C07264=1013.290,308.137,352.891,169.642,52.741,160.224
C07265=1013.283,307.846,352.929,169.634,52.748,160.224
C07266=1013.275,307.555,352.966,169.627,52.756,160.225
C07267=1013.269,307.308,352.997,169.621,52.762,160.225
C07268=1013.263,307.060,353.029,169.613,52.768,160.225
C07269=1013.257,306.812,353.061,169.607,52.774,160.225
C07270=1013.251,306.564,353.092,169.600,52.781,160.225
C07271=1013.245,306.316,353.124,169.594,52.787,160.225
C07272=1013.239,306.069,353.155,169.588,52.793,160.225
C07273=1013.233,305.820,353.186,169.581,52.799,160.225
C07274=1013.227,305.573,353.218,169.575,52.805,160.225
C07275=1013.221,305.325,353.250,169.568,52.812,160.226
C07276=1013.214,305.077,353.281,169.562,52.818,160.226
C07277=1013.209,304.829,353.312,169.556,52.824,160.226
C07278=1013.202,304.581,353.343,169.549,52.830,160.226
C07279=1013.197,304.333,353.375,169.543,52.837,160.226
C07280=1013.190,304.085,353.406,169.536,52.843,160.226
C07281=1013.185,303.837,353.437,169.530,52.849,160.227
C07282=1013.178,303.589,353.469,169.524,52.856,160.227
C07283=1013.173,303.342,353.501,169.517,52.862,160.227
C07284=1013.167,303.093,353.531,169.511,52.868,160.227
C07285=1013.161,302.846,353.563,169.505,52.875,160.227
C07286=1013.155,302.597,353.594,169.498,52.881,160.227
C07287=1013.149,302.350,353.625,169.493,52.887,160.228
C07288=1013.144,302.102,353.656,169.486,52.894,160.228
C07289=1013.138,301.854,353.688,169.480,52.900,160.228
C07290=1013.131,301.607,353.719,169.474,52.906,160.228
C07291=1013.126,301.358,353.750,169.467,52.913,160.228
C07292=1013.120,301.110,353.782,169.461,52.919,160.229
C07293=1013.115,300.862,353.812,169.454,52.926,160.229
C07294=1013.109,300.614,353.843,169.448,52.932,160.229
C07295=1013.103,300.366,353.874,169.442,52.938,160.229
C07296=1013.098,300.118,353.905,169.436,52.945,160.230
C07297=1013.091,299.870,353.937,169.430,52.952,160.230
C07298=1013.086,299.622,353.968,169.423,52.958,160.230
C07299=1013.080,299.374,353.998,169.417,52.964,160.230
C07300=1013.074,299.126,354.030,169.411,52.971,160.230
C07301=1013.068,298.878,354.060,169.404,52.977,160.231
C07302=1013.063,298.631,354.092,169.398,52.984,160.231
C07303=1013.057,298.383,354.122,169.393,52.990,160.231
C07304=1013.051,298.134,354.154,169.386,52.997,160.231
C07305=1013.046,297.886,354.184,169.380,53.004,160.232
C07306=1013.040,297.639,354.216,169.373,53.010,160.232
C07307=1013.034,297.391,354.246,169.368,53.017,160.232
C07308=1013.029,297.142,354.277,169.362,53.023,160.232
C07309=1013.023,296.894,354.308,169.355,53.030,160.233
C07310=1013.017,296.647,354.339,169.349,53.037,160.233
C07311=1013.012,296.399,354.370,169.344,53.043,160.233
C07312=1013.007,296.151,354.401,169.337,53.050,160.233
C07313=1013.000,295.902,354.431,169.331,53.056,160.234
C07314=1012.995,295.654,354.462,169.325,53.063,160.234
C07315=1012.989,295.406,354.493,169.318,53.070,160.234
C07316=1012.984,295.158,354.524,169.313,53.076,160.234
C07317=1012.978,294.911,354.554,169.306,53.083,160.235
C07318=1012.973,294.663,354.586,169.300,53.089,160.235
C07319=1012.967,294.415,354.616,169.294,53.096,160.235
C07320=1012.962,294.167,354.647,169.288,53.103,160.235
C07321=1012.956,293.919,354.677,169.282,53.109,160.236
C07322=1012.951,293.671,354.708,169.276,53.116,160.236
C07323=1012.945,293.398,354.742,169.269,53.123,160.236
C07324=1012.939,293.126,354.776,169.262,53.131,160.237
C07325=1012.933,292.853,354.810,169.256,53.138,160.237
C07326=1012.927,292.582,354.843,169.249,53.145,160.237
C07327=1012.922,292.334,354.874,169.243,53.153,160.238
C07328=1012.916,292.085,354.903,169.237,53.159,160.238
C07329=1012.911,291.837,354.934,169.231,53.166,160.238
C07330=1012.905,291.590,354.964,169.225,53.173,160.239
C07331=1012.899,291.342,354.994,169.219,53.180,160.239
C07332=1012.894,291.093,355.024,169.213,53.187,160.239
C07333=1012.888,290.845,355.055,169.207,53.194,160.240
C07334=1012.883,290.597,355.085,169.200,53.201,160.240
C07335=1012.877,290.349,355.115,169.195,53.208,160.240
C07336=1012.871,290.101,355.145,169.189,53.214,160.241
C07337=1012.866,289.853,355.175,169.183,53.222,160.241
C07338=1012.860,289.605,355.205,169.177,53.228,160.241
C07339=1012.854,289.356,355.235,169.171,53.236,160.242
C07340=1012.849,289.109,355.265,169.165,53.242,160.242
C07341=1012.843,288.860,355.295,169.159,53.250,160.242
C07342=1012.837,288.612,355.325,169.153,53.256,160.243
C07343=1012.832,288.364,355.355,169.147,53.264,160.243
C07344=1012.826,288.115,355.384,169.141,53.270,160.243
C07345=1012.821,287.868,355.414,169.135,53.278,160.244
C07346=1012.816,287.620,355.444,169.130,53.285,160.244
C07347=1012.810,287.372,355.474,169.124,53.292,160.245
C07348=1012.804,287.124,355.504,169.118,53.299,160.245
C07349=1012.799,286.875,355.534,169.112,53.306,160.245
C07350=1012.793,286.627,355.564,169.105,53.313,160.246
C07351=1012.787,286.379,355.594,169.100,53.320,160.246
C07352=1012.782,286.131,355.623,169.094,53.328,160.247
C07353=1012.777,285.883,355.653,169.088,53.334,160.247
C07354=1012.771,285.635,355.683,169.082,53.342,160.247
C07355=1012.766,285.386,355.713,169.077,53.349,160.248
C07356=1012.760,285.138,355.742,169.070,53.356,160.248
C07357=1012.755,284.890,355.771,169.065,53.363,160.248
C07358=1012.750,284.642,355.801,169.058,53.371,160.249
C07359=1012.744,284.393,355.831,169.053,53.378,160.249
C07360=1012.738,284.146,355.861,169.047,53.385,160.250
C07361=1012.733,283.898,355.890,169.041,53.392,160.250
C07362=1012.727,283.650,355.919,169.035,53.400,160.250
C07363=1012.722,283.401,355.949,169.029,53.407,160.251
C07364=1012.717,283.154,355.978,169.023,53.414,160.251
C07365=1012.711,282.905,356.007,169.018,53.421,160.252
C07366=1012.705,282.657,356.037,169.012,53.429,160.252
C07367=1012.700,282.408,356.066,169.006,53.436,160.253
C07368=1012.694,282.160,356.095,169.000,53.444,160.253
C07369=1012.689,281.912,356.124,168.995,53.451,160.254
C07370=1012.683,281.664,356.154,168.988,53.459,160.254
C07371=1012.678,281.416,356.183,168.983,53.466,160.255
C07372=1012.672,281.168,356.212,168.977,53.473,160.255
C07373=1012.666,280.919,356.242,168.972,53.481,160.255
C07374=1012.662,280.671,356.270,168.965,53.488,160.256
C07375=1012.656,280.423,356.299,168.960,53.495,160.256
C07376=1012.651,280.175,356.329,168.954,53.503,160.257
C07377=1012.645,279.927,356.358,168.948,53.510,160.257
C07378=1012.640,279.678,356.387,168.942,53.518,160.258
C07379=1012.634,279.430,356.416,168.936,53.525,160.258
C07380=1012.629,279.182,356.445,168.931,53.533,160.259
C07381=1012.624,278.934,356.475,168.924,53.540,160.259
C07382=1012.618,278.685,356.503,168.920,53.548,160.260
C07383=1012.612,278.425,356.534,168.913,53.556,160.260
C07384=1012.607,278.165,356.565,168.907,53.563,160.260
C07385=1012.602,277.905,356.595,168.901,53.572,160.261
C07386=1012.596,277.645,356.626,168.895,53.579,160.261
C07387=1012.587,277.237,356.672,168.886,53.592,160.262
C07388=1012.579,276.829,356.720,168.877,53.604,160.263
C07389=1012.570,276.422,356.768,168.867,53.617,160.264
C07390=1012.561,276.014,356.816,168.858,53.629,160.265
C07391=1012.347,278.241,356.191,168.878,53.661,160.276
C07392=1012.354,278.605,356.149,168.887,53.650,160.276
C07393=1012.362,278.970,356.107,168.895,53.639,160.275
C07394=1012.370,279.335,356.064,168.904,53.628,160.274
C07395=1012.379,279.699,356.021,168.912,53.617,160.274
C07396=1012.383,279.947,355.992,168.918,53.609,160.273
C07397=1012.389,280.196,355.963,168.923,53.602,160.273
C07398=1012.394,280.443,355.934,168.929,53.594,160.272
C07399=1012.400,280.692,355.904,168.936,53.587,160.272
C07400=1012.404,280.940,355.876,168.941,53.580,160.271
C07401=1012.410,281.189,355.846,168.947,53.572,160.271
C07402=1012.416,281.437,355.817,168.952,53.565,160.270
C07403=1012.421,281.684,355.788,168.959,53.557,160.270
C07404=1012.426,281.934,355.759,168.964,53.550,160.270
C07405=1012.433,282.182,355.730,168.970,53.542,160.269
C07406=1012.437,282.429,355.701,168.977,53.535,160.269
C07407=1012.443,282.678,355.671,168.982,53.528,160.268
C07408=1012.448,282.926,355.641,168.988,53.520,160.268
C07409=1012.454,283.174,355.613,168.993,53.513,160.267
C07410=1012.460,283.422,355.583,169.000,53.505,160.267
C07411=1012.465,283.671,355.553,169.005,53.498,160.266
C07412=1012.471,283.918,355.525,169.011,53.490,160.266
C07413=1012.476,284.166,355.495,169.016,53.483,160.266
C07414=1012.482,284.415,355.466,169.023,53.476,160.265
C07415=1012.487,284.663,355.436,169.028,53.469,160.265
C07416=1012.492,284.911,355.407,169.035,53.462,160.264
C07417=1012.498,285.160,355.377,169.040,53.454,160.264
C07418=1012.503,285.408,355.347,169.047,53.447,160.264
C07419=1012.508,285.656,355.318,169.052,53.440,160.263
C07420=1012.514,285.904,355.288,169.058,53.433,160.263
C07421=1012.519,286.152,355.258,169.065,53.425,160.263
C07422=1012.525,286.400,355.228,169.070,53.419,160.262
C07423=1012.530,286.648,355.199,169.077,53.411,160.262
C07424=1012.535,286.897,355.170,169.082,53.404,160.261
C07425=1012.541,287.144,355.139,169.089,53.397,160.261
C07426=1012.547,287.393,355.110,169.094,53.390,160.261
C07427=1012.552,287.641,355.080,169.100,53.382,160.260
C07428=1012.558,287.889,355.050,169.106,53.376,160.260
C07429=1012.563,288.137,355.020,169.112,53.368,160.260
C07430=1012.568,288.385,354.991,169.118,53.362,160.259
C07431=1012.574,288.633,354.960,169.124,53.354,160.259
C07432=1012.580,288.882,354.931,169.129,53.347,160.258
C07433=1012.585,289.130,354.901,169.136,53.340,160.258
C07434=1012.591,289.378,354.871,169.141,53.333,160.258
C07435=1012.597,289.626,354.841,169.148,53.326,160.258
C07436=1012.602,289.874,354.811,169.154,53.319,160.257
C07437=1012.607,290.122,354.781,169.160,53.312,160.257
C07438=1012.613,290.370,354.751,169.166,53.305,160.256
C07439=1012.619,290.618,354.721,169.172,53.298,160.256
C07440=1012.625,290.866,354.691,169.178,53.291,160.256
C07441=1012.630,291.114,354.661,169.183,53.284,160.255
C07442=1012.635,291.362,354.631,169.190,53.277,160.255
C07443=1012.641,291.610,354.600,169.195,53.270,160.255
C07444=1012.646,291.859,354.571,169.202,53.263,160.254
C07445=1012.652,292.107,354.540,169.207,53.256,160.254
C07446=1012.658,292.354,354.510,169.214,53.249,160.254
C07447=1012.663,292.603,354.479,169.220,53.243,160.253
C07448=1012.669,292.877,354.445,169.227,53.235,160.253
C07449=1012.676,293.152,354.412,169.234,53.227,160.253
C07450=1012.681,293.426,354.378,169.240,53.220,160.253
C07451=1012.688,293.701,354.344,169.248,53.213,160.252
C07452=1012.693,293.949,354.313,169.253,53.206,160.252
C07453=1012.699,294.197,354.283,169.259,53.199,160.251
C07454=1012.704,294.445,354.252,169.265,53.192,160.251
C07455=1012.710,294.693,354.221,169.271,53.186,160.251
C07456=1012.715,294.941,354.190,169.278,53.179,160.251
C07457=1012.720,295.189,354.160,169.284,53.172,160.251
C07458=1012.726,295.437,354.129,169.290,53.166,160.250
C07459=1012.731,295.685,354.099,169.296,53.159,160.250
C07460=1012.736,295.933,354.068,169.302,53.153,160.250
C07461=1012.742,296.181,354.037,169.309,53.146,160.250
C07462=1012.747,296.429,354.006,169.314,53.139,160.249
C07463=1012.754,296.677,353.976,169.321,53.132,160.249
C07464=1012.759,296.925,353.944,169.327,53.125,160.249
C07465=1012.765,297.173,353.914,169.332,53.119,160.248
C07466=1012.770,297.421,353.883,169.339,53.112,160.248
C07467=1012.775,297.669,353.852,169.345,53.105,160.248
C07468=1012.781,297.917,353.821,169.352,53.099,160.248
C07469=1012.787,298.165,353.789,169.357,53.092,160.247
C07470=1012.793,298.413,353.759,169.364,53.086,160.247
C07471=1012.798,298.661,353.728,169.370,53.080,160.247
C07472=1012.804,298.909,353.698,169.376,53.073,160.247
C07473=1012.810,299.157,353.666,169.383,53.066,160.247
C07474=1012.815,299.405,353.635,169.389,53.060,160.246
C07475=1012.820,299.653,353.604,169.396,53.053,160.246
C07476=1012.827,299.900,353.573,169.401,53.047,160.246
C07477=1012.832,300.149,353.542,169.407,53.040,160.246
C07478=1012.838,300.397,353.512,169.414,53.033,160.245
C07479=1012.843,300.644,353.480,169.420,53.027,160.245
C07480=1012.850,300.893,353.449,169.427,53.021,160.245
C07481=1012.855,301.140,353.418,169.433,53.014,160.245
C07482=1012.861,301.388,353.387,169.439,53.007,160.245
C07483=1012.867,301.637,353.356,169.445,53.001,160.244
C07484=1012.873,301.884,353.325,169.451,52.995,160.244
C07485=1012.878,302.132,353.294,169.458,52.988,160.244
C07486=1012.885,302.380,353.263,169.464,52.982,160.244
C07487=1012.890,302.628,353.232,169.471,52.976,160.244
C07488=1012.897,302.876,353.200,169.477,52.969,160.244
C07489=1012.902,303.124,353.169,169.484,52.962,160.243
C07490=1012.908,303.372,353.138,169.490,52.956,160.243
C07491=1012.914,303.620,353.106,169.497,52.950,160.243
C07492=1012.920,303.868,353.076,169.503,52.943,160.243
C07493=1012.926,304.116,353.044,169.509,52.938,160.243
C07494=1012.932,304.363,353.013,169.516,52.931,160.243
C07495=1012.937,304.612,352.981,169.521,52.924,160.242
C07496=1012.943,304.859,352.950,169.529,52.918,160.242
C07497=1012.949,305.107,352.918,169.534,52.912,160.242
C07498=1012.955,305.355,352.887,169.542,52.906,160.242
C07499=1012.961,305.603,352.856,169.547,52.899,160.242
C07500=1012.967,305.851,352.824,169.554,52.893,160.242
C07501=1012.973,306.099,352.793,169.560,52.887,160.242
C07502=1012.979,306.348,352.762,169.566,52.880,160.241
C07503=1012.985,306.595,352.730,169.573,52.874,160.241
C07504=1012.991,306.843,352.698,169.579,52.868,160.241
C07505=1012.997,307.090,352.667,169.586,52.862,160.241
C07506=1013.003,307.338,352.635,169.593,52.856,160.241
C07507=1013.010,307.587,352.605,169.599,52.849,160.241
C07508=1013.016,307.879,352.566,169.607,52.842,160.241
C07509=1013.024,308.172,352.530,169.615,52.835,160.241
C07510=1013.031,308.464,352.493,169.623,52.828,160.240
C07511=1013.038,308.757,352.456,169.630,52.820,160.240
C07512=1013.044,309.004,352.423,169.636,52.814,160.240
C07513=1013.050,309.252,352.391,169.643,52.808,160.240
C07514=1013.056,309.501,352.359,169.650,52.802,160.240
C07515=1013.061,309.748,352.327,169.656,52.796,160.240
C07516=1013.068,309.996,352.295,169.663,52.790,160.240
C07517=1013.072,310.244,352.262,169.669,52.784,160.240
C07518=1013.079,310.491,352.230,169.675,52.778,160.240
C07519=1013.085,310.739,352.198,169.683,52.772,160.240
C07520=1013.090,310.987,352.166,169.689,52.766,160.240
C07521=1013.096,311.235,352.133,169.695,52.761,160.239
C07522=1013.102,311.483,352.101,169.702,52.754,160.239
C07523=1013.108,311.731,352.068,169.709,52.749,160.239
C07524=1013.113,311.978,352.036,169.715,52.743,160.239
C07525=1013.120,312.226,352.004,169.722,52.737,160.239
C07526=1013.126,312.474,351.971,169.728,52.731,160.239
C07527=1013.132,312.722,351.939,169.735,52.725,160.239
C07528=1013.137,312.969,351.907,169.742,52.719,160.239
C07529=1013.143,313.217,351.874,169.748,52.714,160.239
C07530=1013.149,313.465,351.841,169.755,52.708,160.239
C07531=1013.155,313.713,351.809,169.762,52.702,160.239
C07532=1013.161,313.960,351.776,169.768,52.696,160.239
C07533=1013.168,314.208,351.743,169.775,52.690,160.239
C07534=1013.173,314.455,351.712,169.781,52.684,160.239
C07535=1013.179,314.703,351.678,169.789,52.678,160.239
C07536=1013.185,314.951,351.646,169.795,52.673,160.239
C07537=1013.191,315.199,351.614,169.802,52.667,160.239
C07538=1013.197,315.447,351.581,169.809,52.661,160.239
C07539=1013.203,315.694,351.548,169.815,52.656,160.239
C07540=1013.209,315.942,351.515,169.821,52.650,160.239
C07541=1013.215,316.190,351.483,169.829,52.644,160.239
C07542=1013.221,316.438,351.450,169.835,52.639,160.239
C07543=1013.228,316.686,351.417,169.842,52.633,160.239
C07544=1013.234,316.933,351.385,169.849,52.627,160.239
C07545=1013.240,317.181,351.352,169.855,52.622,160.239
C07546=1013.246,317.429,351.319,169.863,52.616,160.239
C07547=1013.252,317.677,351.287,169.869,52.610,160.239
C07548=1013.258,317.925,351.254,169.877,52.605,160.239
C07549=1013.264,318.172,351.221,169.883,52.599,160.239
C07550=1013.271,318.420,351.188,169.890,52.593,160.239
C07551=1013.276,318.668,351.155,169.897,52.588,160.239
C07552=1013.282,318.915,351.122,169.903,52.582,160.239
C07553=1013.289,319.163,351.089,169.910,52.576,160.239
C07554=1013.296,319.411,351.056,169.917,52.571,160.239
C07555=1013.302,319.659,351.024,169.924,52.565,160.239
C07556=1013.307,319.907,350.990,169.931,52.560,160.240
C07557=1013.314,320.154,350.958,169.937,52.554,160.239
C07558=1013.320,320.401,350.924,169.945,52.549,160.240
C07559=1013.327,320.649,350.891,169.951,52.543,160.240
C07560=1013.334,320.897,350.858,169.959,52.538,160.240
C07561=1013.339,321.145,350.825,169.965,52.532,160.240
C07562=1013.345,321.393,350.792,169.973,52.526,160.240
C07563=1013.352,321.640,350.759,169.979,52.521,160.240
C07564=1013.359,321.888,350.726,169.987,52.515,160.240
C07565=1013.365,322.135,350.693,169.993,52.510,160.240
C07566=1013.371,322.383,350.660,170.000,52.505,160.240
C07567=1013.377,322.631,350.627,170.007,52.499,160.240
C07568=1013.385,322.929,350.587,170.016,52.493,160.241
C07569=1013.393,323.227,350.547,170.024,52.486,160.241
C07570=1013.401,323.525,350.507,170.032,52.480,160.241
C07571=1013.409,323.824,350.467,170.041,52.473,160.241
C07572=1013.415,324.072,350.433,170.048,52.468,160.241
C07573=1013.421,324.319,350.400,170.055,52.462,160.241
C07574=1013.428,324.567,350.367,170.062,52.457,160.241
C07575=1013.435,324.814,350.334,170.070,52.451,160.241
C07576=1013.441,325.061,350.301,170.076,52.446,160.242
C07577=1013.447,325.310,350.267,170.083,52.441,160.241
C07578=1013.454,325.557,350.233,170.090,52.435,160.242
C07579=1013.461,325.805,350.200,170.097,52.430,160.242
C07580=1013.467,326.053,350.166,170.105,52.425,160.242
C07581=1013.473,326.300,350.132,170.112,52.420,160.242
C07582=1013.480,326.548,350.098,170.119,52.414,160.242
C07583=1013.486,326.795,350.064,170.126,52.409,160.243
C07584=1013.493,327.043,350.031,170.133,52.404,160.243
C07585=1013.498,327.290,349.997,170.140,52.399,160.243
C07586=1013.505,327.538,349.963,170.147,52.394,160.243
C07587=1013.511,327.785,349.929,170.155,52.389,160.243
C07588=1013.518,328.033,349.895,170.161,52.384,160.243
C07589=1013.524,328.281,349.861,170.169,52.378,160.244
C07590=1013.531,328.528,349.827,170.176,52.373,160.244
C07591=1013.537,328.776,349.793,170.183,52.369,160.244
C07592=1013.543,329.024,349.758,170.191,52.363,160.244
C07593=1013.551,329.271,349.725,170.197,52.358,160.244
C07594=1013.556,329.519,349.691,170.205,52.353,160.245
C07595=1013.563,329.767,349.656,170.212,52.348,160.245
C07596=1013.569,330.014,349.623,170.219,52.343,160.245
C07597=1013.576,330.262,349.588,170.227,52.338,160.245
C07598=1013.582,330.509,349.554,170.234,52.333,160.246
C07599=1013.589,330.756,349.520,170.241,52.328,160.246
C07600=1013.595,331.004,349.486,170.249,52.322,160.246
C07601=1013.602,331.252,349.452,170.256,52.318,160.246
C07602=1013.609,331.499,349.417,170.264,52.313,160.247
C07603=1013.615,331.747,349.383,170.270,52.308,160.247
C07604=1013.622,331.995,349.349,170.277,52.303,160.247
C07605=1013.628,332.243,349.314,170.285,52.298,160.247
C07606=1013.635,332.489,349.280,170.292,52.294,160.248
C07607=1013.642,332.737,349.246,170.300,52.288,160.248
C07608=1013.648,332.984,349.210,170.307,52.283,160.248
C07609=1013.655,333.232,349.176,170.315,52.279,160.248
C07610=1013.661,333.480,349.142,170.321,52.274,160.248
C07611=1013.667,333.727,349.107,170.330,52.269,160.249
C07612=1013.674,333.975,349.072,170.337,52.264,160.249
C07613=1013.681,334.222,349.037,170.344,52.259,160.249
C07614=1013.687,334.470,349.003,170.352,52.255,160.250
C07615=1013.694,334.718,348.968,170.358,52.250,160.250
C07616=1013.700,334.964,348.933,170.366,52.245,160.250
C07617=1013.707,335.212,348.899,170.373,52.240,160.250
C07618=1013.714,335.459,348.864,170.381,52.235,160.251
C07619=1013.720,335.707,348.830,170.388,52.231,160.251
C07620=1013.727,335.955,348.794,170.396,52.226,160.251
C07621=1013.734,336.202,348.759,170.403,52.221,160.252
C07622=1013.740,336.450,348.725,170.411,52.217,160.252
C07623=1013.747,336.698,348.690,170.418,52.212,160.253
C07624=1013.754,336.945,348.655,170.426,52.207,160.253
C07625=1013.761,337.192,348.619,170.433,52.202,160.253
C07626=1013.768,337.440,348.584,170.441,52.198,160.254
C07627=1013.774,337.688,348.550,170.449,52.193,160.254
C07628=1013.782,337.981,348.509,170.458,52.187,160.254
C07629=1013.790,338.275,348.467,170.467,52.182,160.255
C07630=1013.798,338.568,348.425,170.476,52.176,160.255
C07631=1013.807,338.863,348.383,170.485,52.171,160.256
C07632=1013.813,339.110,348.348,170.492,52.167,160.256
C07633=1013.819,339.358,348.312,170.500,52.162,160.256
C07634=1013.826,339.605,348.277,170.507,52.157,160.257
C07635=1013.833,339.852,348.242,170.515,52.153,160.257
C07636=1013.840,340.100,348.207,170.522,52.148,160.257
C07637=1013.847,340.347,348.172,170.531,52.144,160.258
C07638=1013.854,340.594,348.136,170.538,52.140,160.258
C07639=1013.860,340.842,348.100,170.546,52.135,160.259
C07640=1013.867,341.090,348.065,170.554,52.130,160.259
C07641=1013.874,341.337,348.030,170.562,52.126,160.260
C07642=1013.881,341.584,347.994,170.570,52.121,160.260
C07643=1013.888,341.831,347.959,170.577,52.117,160.260
C07644=1013.894,342.079,347.923,170.585,52.112,160.261
C07645=1013.901,342.326,347.887,170.593,52.109,160.261
C07646=1013.908,342.574,347.852,170.601,52.104,160.262
C07647=1013.915,342.821,347.816,170.608,52.100,160.262
C07648=1013.922,343.069,347.780,170.616,52.095,160.262
C07649=1013.929,343.316,347.744,170.624,52.091,160.263
C07650=1013.936,343.563,347.709,170.632,52.086,160.263
C07651=1013.942,343.810,347.673,170.640,52.082,160.264
C07652=1013.949,344.058,347.637,170.647,52.078,160.264
C07653=1013.956,344.305,347.602,170.656,52.073,160.265
C07654=1013.963,344.552,347.566,170.663,52.069,160.265
C07655=1013.971,344.799,347.529,170.671,52.065,160.266
C07656=1013.977,345.047,347.494,170.678,52.061,160.266
C07657=1013.985,345.295,347.458,170.686,52.056,160.267
C07658=1013.992,345.541,347.422,170.695,52.052,160.267
C07659=1013.998,345.789,347.387,170.702,52.048,160.268
C07660=1014.005,346.036,347.350,170.711,52.044,160.268
C07661=1014.012,346.283,347.314,170.718,52.039,160.269
C07662=1014.020,346.531,347.278,170.726,52.035,160.269
C07663=1014.026,346.778,347.242,170.735,52.030,160.270
C07664=1014.034,347.026,347.206,170.742,52.027,160.270
C07665=1014.040,347.273,347.169,170.751,52.023,160.271
C07666=1014.048,347.520,347.133,170.758,52.018,160.271
C07667=1014.054,347.767,347.097,170.766,52.014,160.272
C07668=1014.062,348.015,347.060,170.775,52.010,160.272
C07669=1014.068,348.262,347.024,170.782,52.006,160.273
C07670=1014.076,348.509,346.988,170.791,52.002,160.273
C07671=1014.082,348.756,346.951,170.799,51.998,160.274
C07672=1014.090,349.004,346.915,170.807,51.994,160.275
C07673=1014.097,349.251,346.878,170.815,51.989,160.275
C07674=1014.104,349.498,346.842,170.823,51.986,160.276
C07675=1014.111,349.745,346.805,170.831,51.982,160.276
C07676=1014.118,349.992,346.769,170.840,51.978,160.277
C07677=1014.125,350.240,346.732,170.847,51.974,160.277
C07678=1014.133,350.487,346.695,170.856,51.970,160.278
C07679=1014.139,350.734,346.659,170.864,51.966,160.279
C07680=1014.147,350.981,346.623,170.871,51.962,160.279
C07681=1014.154,351.229,346.586,170.880,51.958,160.280
C07682=1014.161,351.476,346.548,170.889,51.954,160.280
C07683=1014.168,351.723,346.512,170.896,51.950,160.281
C07684=1014.175,351.971,346.476,170.905,51.946,160.281
C07685=1014.183,352.217,346.439,170.913,51.942,160.282
C07686=1014.190,352.465,346.402,170.922,51.938,160.283
C07687=1014.198,352.711,346.365,170.929,51.934,160.283
C07688=1014.206,353.003,346.321,170.940,51.929,160.284
C07689=1014.215,353.294,346.278,170.950,51.925,160.285
C07690=1014.223,353.586,346.234,170.959,51.920,160.286
C07691=1014.232,353.877,346.191,170.969,51.916,160.286
C07692=1014.239,354.124,346.154,170.978,51.913,160.287
C07693=1014.246,354.372,346.117,170.986,51.908,160.288
C07694=1014.254,354.618,346.080,170.994,51.905,160.288
C07695=1014.261,354.865,346.043,171.002,51.901,160.289
C07696=1014.268,355.112,346.005,171.011,51.897,160.290
C07697=1014.275,355.359,345.968,171.020,51.893,160.290
C07698=1014.283,355.607,345.931,171.027,51.890,160.291
C07699=1014.290,355.854,345.894,171.036,51.886,160.292
C07700=1014.298,356.101,345.856,171.045,51.882,160.292
C07701=1014.306,356.348,345.819,171.053,51.878,160.293
C07702=1014.313,356.595,345.782,171.061,51.875,160.294
C07703=1014.320,356.842,345.744,171.070,51.871,160.294
C07704=1014.327,357.089,345.707,171.079,51.868,160.295
C07705=1014.335,357.336,345.669,171.088,51.864,160.296
C07706=1014.343,357.583,345.632,171.097,51.860,160.297
C07707=1014.350,357.831,345.595,171.104,51.857,160.297
C07708=1014.358,358.078,345.557,171.113,51.853,160.298
C07709=1014.365,358.325,345.519,171.122,51.850,160.299
C07710=1014.373,358.571,345.482,171.131,51.846,160.300
C07711=1014.380,358.818,345.444,171.140,51.842,160.301
C07712=1014.388,359.066,345.407,171.147,51.839,160.301
C07713=1014.395,359.312,345.369,171.156,51.835,160.302
C07714=1014.402,359.559,345.331,171.165,51.832,160.303
C07715=1014.410,359.807,345.293,171.174,51.828,160.304
C07716=1014.417,360.054,345.254,171.183,51.824,160.304
C07717=1014.424,360.301,345.217,171.191,51.821,160.305
C07718=1014.432,360.548,345.179,171.200,51.818,160.306
C07719=1014.439,360.795,345.141,171.209,51.815,160.307
C07720=1014.447,361.042,345.102,171.218,51.811,160.308
C07721=1014.455,361.289,345.065,171.227,51.808,160.308
C07722=1014.462,361.536,345.027,171.236,51.804,160.309
C07723=1014.470,361.782,344.988,171.243,51.801,160.310
C07724=1014.478,362.030,344.950,171.252,51.797,160.311
C07725=1014.485,362.276,344.912,171.261,51.794,160.311
C07726=1014.493,362.523,344.874,171.270,51.790,160.312
C07727=1014.500,362.771,344.836,171.279,51.787,160.313
C07728=1014.508,363.017,344.798,171.288,51.784,160.314
C07729=1014.516,363.264,344.759,171.297,51.780,160.315
C07730=1014.524,363.511,344.721,171.306,51.777,160.316
C07731=1014.531,363.758,344.683,171.315,51.774,160.317
C07732=1014.539,364.005,344.645,171.324,51.771,160.318
C07733=1014.547,364.252,344.607,171.332,51.768,160.318
C07734=1014.555,364.499,344.568,171.341,51.764,160.319
C07735=1014.562,364.746,344.530,171.350,51.761,160.320
C07736=1014.571,364.993,344.491,171.359,51.757,160.321
C07737=1014.578,365.239,344.453,171.369,51.755,160.322
C07738=1014.586,365.487,344.414,171.378,51.751,160.323
C07739=1014.593,365.733,344.375,171.387,51.748,160.324
C07740=1014.601,365.981,344.337,171.396,51.745,160.325
C07741=1014.609,366.228,344.298,171.405,51.742,160.325
C07742=1014.617,366.474,344.260,171.414,51.738,160.326
C07743=1014.625,366.722,344.221,171.423,51.735,160.327
C07744=1014.633,366.967,344.182,171.432,51.732,160.328
C07745=1014.641,367.215,344.144,171.441,51.729,160.329
C07746=1014.649,367.462,344.105,171.451,51.726,160.330
C07747=1014.656,367.708,344.066,171.460,51.722,160.331
C07748=1014.666,368.007,344.019,171.471,51.719,160.332
C07749=1014.675,368.306,343.971,171.482,51.715,160.333
C07750=1014.685,368.605,343.925,171.494,51.712,160.335
C07751=1014.694,368.903,343.876,171.505,51.708,160.336
C07752=1014.702,369.151,343.838,171.514,51.705,160.337
C07753=1014.711,369.397,343.798,171.524,51.702,160.338
C07754=1014.718,369.643,343.759,171.533,51.699,160.339
C07755=1014.726,369.891,343.720,171.542,51.696,160.340
C07756=1014.734,370.138,343.680,171.551,51.693,160.341
C07757=1014.742,370.384,343.641,171.561,51.690,160.342
C07758=1014.750,370.631,343.602,171.570,51.688,160.343
C07759=1014.758,370.878,343.562,171.580,51.684,160.344
C07760=1014.766,371.124,343.524,171.590,51.681,160.345
C07761=1014.775,371.371,343.484,171.599,51.678,160.346
C07762=1014.782,371.618,343.444,171.608,51.676,160.347
C07763=1014.790,371.865,343.406,171.618,51.673,160.348
C07764=1014.798,372.112,343.366,171.627,51.670,160.349
C07765=1014.807,372.358,343.326,171.636,51.667,160.350
C07766=1014.815,372.605,343.287,171.646,51.664,160.351
C07767=1014.823,372.852,343.247,171.656,51.661,160.352
C07768=1014.831,373.099,343.208,171.666,51.658,160.353
C07769=1014.840,373.345,343.169,171.675,51.656,160.354
C07770=1014.847,373.592,343.129,171.684,51.653,160.356
C07771=1014.856,373.838,343.089,171.694,51.650,160.357
C07772=1014.864,374.085,343.049,171.704,51.647,160.358
C07773=1014.872,374.331,343.009,171.714,51.644,160.359
C07774=1014.881,374.578,342.970,171.723,51.642,160.360
C07775=1014.889,374.826,342.930,171.733,51.639,160.361
C07776=1014.898,375.072,342.890,171.743,51.636,160.362
C07777=1014.906,375.319,342.850,171.753,51.633,160.363
C07778=1014.914,375.565,342.810,171.762,51.631,160.365
C07779=1014.922,375.811,342.770,171.772,51.628,160.366
C07780=1014.930,376.058,342.730,171.782,51.625,160.367
C07781=1014.939,376.305,342.689,171.792,51.623,160.368
C07782=1014.947,376.552,342.650,171.801,51.620,160.369
C07783=1014.955,376.798,342.609,171.811,51.618,160.370
C07784=1014.963,377.044,342.568,171.822,51.615,160.372
C07785=1014.971,377.291,342.529,171.831,51.613,160.373
C07786=1014.980,377.538,342.488,171.841,51.610,160.374
C07787=1014.988,377.784,342.447,171.852,51.607,160.375
C07788=1014.997,378.030,342.407,171.861,51.605,160.376
C07789=1015.005,378.278,342.367,171.871,51.603,160.378
C07790=1015.013,378.524,342.326,171.882,51.600,160.379
C07791=1015.021,378.771,342.286,171.891,51.598,160.380
C07792=1015.031,379.017,342.245,171.901,51.595,160.381
C07793=1015.039,379.263,342.205,171.911,51.592,160.383
C07794=1015.047,379.510,342.164,171.921,51.590,160.384
C07795=1015.056,379.756,342.124,171.931,51.588,160.385
C07796=1015.064,380.003,342.083,171.941,51.585,160.386
C07797=1015.073,380.250,342.042,171.951,51.583,160.387
C07798=1015.081,380.496,342.001,171.962,51.580,160.389
C07799=1015.090,380.743,341.961,171.972,51.578,160.390
C07800=1015.098,380.989,341.920,171.983,51.576,160.391
C07801=1015.107,381.236,341.879,171.992,51.573,160.393
C07802=1015.116,381.482,341.838,172.002,51.571,160.394
C07803=1015.124,381.728,341.798,172.013,51.569,160.395
C07804=1015.133,381.975,341.757,172.023,51.567,160.397
C07805=1015.141,382.222,341.716,172.034,51.564,160.398
C07806=1015.151,382.468,341.675,172.043,51.562,160.399
C07807=1015.159,382.715,341.634,172.054,51.559,160.401
C07808=1015.170,383.036,341.580,172.067,51.557,160.402
C07809=1015.182,383.357,341.527,172.082,51.553,160.404
C07810=1015.193,383.679,341.473,172.095,51.551,160.406
C07811=1015.205,384.000,341.420,172.109,51.547,160.408
C07812=1015.214,384.247,341.379,172.119,51.546,160.409
C07813=1015.223,384.494,341.338,172.130,51.543,160.410
C07814=1015.232,384.740,341.296,172.140,51.540,160.412
C07815=1015.241,384.987,341.254,172.151,51.539,160.413
C07816=1015.249,385.232,341.213,172.161,51.536,160.415
C07817=1015.258,385.479,341.172,172.172,51.535,160.416
C07818=1015.267,385.726,341.130,172.182,51.532,160.417
C07819=1015.276,385.972,341.088,172.194,51.530,160.419
C07820=1015.284,386.218,341.047,172.203,51.528,160.420
C07821=1015.293,386.465,341.005,172.215,51.526,160.422
C07822=1015.303,386.711,340.964,172.225,51.524,160.423
C07823=1015.312,386.957,340.922,172.236,51.522,160.425
C07824=1015.321,387.203,340.880,172.247,51.520,160.426
C07825=1015.330,387.450,340.839,172.258,51.517,160.428
C07826=1015.339,387.696,340.797,172.268,51.516,160.429
C07827=1015.347,387.942,340.754,172.279,51.514,160.431
C07828=1015.356,388.189,340.712,172.290,51.512,160.432
C07829=1015.365,388.435,340.671,172.301,51.509,160.434
C07830=1015.374,388.681,340.629,172.311,51.508,160.435
C07831=1015.383,388.927,340.586,172.322,51.506,160.437
C07832=1015.392,389.173,340.545,172.334,51.504,160.438
C07833=1015.401,389.419,340.502,172.345,51.502,160.440
C07834=1015.410,389.665,340.461,172.355,51.500,160.441
C07835=1015.420,389.911,340.418,172.366,51.498,160.443
C07836=1015.428,390.159,340.375,172.377,51.497,160.444
C07837=1015.438,390.404,340.333,172.389,51.495,160.446
C07838=1015.447,390.651,340.291,172.400,51.493,160.448
C07839=1015.456,390.896,340.249,172.411,51.491,160.449
C07840=1015.466,391.143,340.206,172.423,51.489,160.451
C07841=1015.475,391.389,340.164,172.433,51.488,160.452
C07842=1015.484,391.635,340.122,172.444,51.486,160.454
C07843=1015.494,391.881,340.079,172.455,51.484,160.456
C07844=1015.502,392.128,340.036,172.466,51.482,160.457
C07845=1015.511,392.374,339.994,172.478,51.480,160.459
C07846=1015.521,392.620,339.952,172.489,51.479,160.460
C07847=1015.530,392.866,339.909,172.501,51.477,160.462
C07848=1015.539,393.112,339.866,172.512,51.475,160.464
C07849=1015.549,393.358,339.823,172.523,51.473,160.465
C07850=1015.557,393.604,339.780,172.535,51.472,160.467
C07851=1015.567,393.850,339.737,172.546,51.470,160.469
C07852=1015.576,394.096,339.694,172.558,51.469,160.470
C07853=1015.586,394.343,339.652,172.569,51.467,160.472
C07854=1015.595,394.589,339.609,172.581,51.465,160.474
C07855=1015.605,394.835,339.565,172.592,51.464,160.476
C07856=1015.614,395.080,339.523,172.604,51.462,160.477
C07857=1015.623,395.327,339.479,172.615,51.460,160.479
C07858=1015.633,395.573,339.436,172.627,51.459,160.481
C07859=1015.643,395.819,339.393,172.638,51.458,160.483
C07860=1015.653,396.065,339.350,172.650,51.456,160.484
C07861=1015.662,396.311,339.306,172.661,51.454,160.486
C07862=1015.671,396.557,339.264,172.674,51.453,160.488
C07863=1015.681,396.803,339.220,172.685,51.451,160.490
C07864=1015.691,397.049,339.176,172.697,51.450,160.491
C07865=1015.700,397.295,339.134,172.708,51.449,160.493
C07866=1015.709,397.541,339.090,172.720,51.447,160.495
C07867=1015.720,397.787,339.046,172.732,51.446,160.497
C07868=1015.736,398.202,338.973,172.752,51.443,160.500
C07869=1015.751,398.617,338.899,172.772,51.441,160.503
C07870=1015.398,396.589,338.913,172.658,51.516,160.502
C07871=1015.388,396.343,338.956,172.647,51.518,160.501
C07872=1015.379,396.096,339.000,172.635,51.520,160.499
C07873=1015.369,395.851,339.043,172.622,51.522,160.497
C07874=1015.359,395.605,339.086,172.611,51.523,160.495
C07875=1015.349,395.359,339.129,172.600,51.525,160.494
C07876=1015.341,395.113,339.172,172.588,51.526,160.492
C07877=1015.331,394.867,339.215,172.577,51.528,160.490
C07878=1015.322,394.621,339.257,172.565,51.530,160.488
C07879=1015.312,394.375,339.301,172.554,51.531,160.487
C07880=1015.303,394.129,339.344,172.542,51.533,160.485
C07881=1015.293,393.883,339.387,172.531,51.534,160.483
C07882=1015.284,393.637,339.429,172.519,51.537,160.482
C07883=1015.275,393.390,339.472,172.507,51.539,160.480
C07884=1015.266,393.144,339.515,172.496,51.540,160.478
C07885=1015.256,392.899,339.557,172.484,51.542,160.477
C07886=1015.247,392.652,339.601,172.473,51.544,160.475
C07887=1015.238,392.406,339.643,172.462,51.545,160.473
C07888=1015.229,392.160,339.686,172.450,51.547,160.472
C07889=1015.219,391.914,339.728,172.439,51.549,160.470
C07890=1015.211,391.667,339.771,172.429,51.550,160.468
C07891=1015.201,391.421,339.813,172.417,51.552,160.467
C07892=1015.192,391.175,339.856,172.406,51.554,160.465
C07893=1015.183,390.929,339.898,172.395,51.556,160.464
C07894=1015.173,390.683,339.940,172.384,51.558,160.462
C07895=1015.164,390.437,339.983,172.373,51.560,160.461
C07896=1015.155,390.190,340.025,172.361,51.562,160.459
C07897=1015.145,389.944,340.067,172.350,51.564,160.457
C07898=1015.137,389.698,340.109,172.339,51.566,160.456
C07899=1015.128,389.452,340.152,172.328,51.568,160.454
C07900=1015.119,389.206,340.194,172.317,51.570,160.453
C07901=1015.110,388.959,340.235,172.307,51.572,160.451
C07902=1015.101,388.713,340.278,172.296,51.574,160.450
C07903=1015.092,388.467,340.319,172.284,51.576,160.448
C07904=1015.083,388.221,340.361,172.273,51.578,160.447
C07905=1015.074,387.974,340.403,172.262,51.580,160.445
C07906=1015.065,387.729,340.445,172.252,51.582,160.444
C07907=1015.056,387.482,340.487,172.241,51.584,160.442
C07908=1015.047,387.236,340.529,172.230,51.586,160.441
C07909=1015.038,386.989,340.570,172.219,51.589,160.439
C07910=1015.029,386.743,340.612,172.209,51.590,160.438
C07911=1015.020,386.497,340.654,172.198,51.593,160.436
C07912=1015.011,386.250,340.696,172.187,51.595,160.435
C07913=1015.002,386.004,340.737,172.176,51.598,160.434
C07914=1014.993,385.758,340.779,172.166,51.599,160.432
C07915=1014.985,385.511,340.820,172.155,51.602,160.431
C07916=1014.976,385.265,340.861,172.144,51.604,160.429
C07917=1014.968,385.019,340.903,172.134,51.606,160.428
C07918=1014.959,384.772,340.945,172.123,51.608,160.426
C07919=1014.950,384.525,340.986,172.112,51.611,160.425
C07920=1014.941,384.279,341.027,172.102,51.613,160.424
C07921=1014.932,384.033,341.068,172.091,51.615,160.422
C07922=1014.923,383.787,341.109,172.081,51.618,160.421
C07923=1014.915,383.537,341.151,172.071,51.620,160.420
C07924=1014.906,383.289,341.191,172.060,51.622,160.418
C07925=1014.897,383.040,341.234,172.049,51.625,160.417
C07926=1014.888,382.792,341.274,172.039,51.627,160.415
C07927=1014.879,382.545,341.315,172.028,51.629,160.414
C07928=1014.871,382.299,341.357,172.018,51.631,160.413
C07929=1014.862,382.052,341.398,172.008,51.634,160.411
C07930=1014.853,381.806,341.438,171.997,51.636,160.410
C07931=1014.845,381.559,341.479,171.987,51.639,160.409
C07932=1014.836,381.312,341.520,171.977,51.642,160.408
C07933=1014.827,381.067,341.561,171.967,51.644,160.406
C07934=1014.818,380.820,341.602,171.956,51.646,160.405
C07935=1014.810,380.574,341.642,171.946,51.649,160.404
C07936=1014.801,380.327,341.683,171.935,51.651,160.402
C07937=1014.793,380.081,341.723,171.926,51.653,160.401
C07938=1014.784,379.834,341.764,171.915,51.657,160.400
C07939=1014.776,379.587,341.805,171.905,51.659,160.399
C07940=1014.767,379.341,341.845,171.895,51.661,160.397
C07941=1014.759,379.094,341.886,171.885,51.664,160.396
C07942=1014.751,378.848,341.927,171.875,51.666,160.395
C07943=1014.742,378.601,341.966,171.865,51.669,160.394
C07944=1014.734,378.355,342.007,171.855,51.672,160.393
C07945=1014.726,378.108,342.048,171.844,51.674,160.391
C07946=1014.717,377.861,342.089,171.835,51.677,160.390
C07947=1014.709,377.615,342.128,171.825,51.679,160.389
C07948=1014.701,377.368,342.169,171.815,51.682,160.388
C07949=1014.693,377.122,342.209,171.805,51.684,160.386
C07950=1014.684,376.875,342.249,171.796,51.687,160.385
C07951=1014.676,376.629,342.289,171.785,51.690,160.384
C07952=1014.667,376.382,342.330,171.775,51.693,160.383
C07953=1014.660,376.135,342.370,171.766,51.695,160.382
C07954=1014.651,375.889,342.410,171.755,51.698,160.381
C07955=1014.643,375.643,342.450,171.746,51.701,160.380
C07956=1014.635,375.396,342.491,171.736,51.704,160.378
C07957=1014.626,375.149,342.530,171.726,51.706,160.377
C07958=1014.618,374.902,342.570,171.716,51.709,160.376
C07959=1014.610,374.655,342.610,171.707,51.712,160.375
C07960=1014.602,374.409,342.649,171.697,51.715,160.374
C07961=1014.594,374.163,342.690,171.687,51.718,160.373
C07962=1014.585,373.916,342.729,171.678,51.720,160.372
C07963=1014.577,373.669,342.768,171.668,51.723,160.371
C07964=1014.569,373.422,342.808,171.658,51.726,160.370
C07965=1014.560,373.176,342.847,171.649,51.729,160.368
C07966=1014.553,372.929,342.887,171.639,51.732,160.367
C07967=1014.544,372.682,342.927,171.630,51.735,160.366
C07968=1014.536,372.436,342.966,171.619,51.738,160.365
C07969=1014.528,372.189,343.006,171.610,51.741,160.364
C07970=1014.520,371.942,343.045,171.601,51.744,160.363
C07971=1014.511,371.695,343.084,171.591,51.746,160.362
C07972=1014.504,371.448,343.124,171.581,51.749,160.361
C07973=1014.495,371.202,343.163,171.572,51.753,160.360
C07974=1014.488,370.955,343.203,171.562,51.756,160.359
C07975=1014.479,370.708,343.242,171.553,51.758,160.358
C07976=1014.472,370.462,343.281,171.544,51.761,160.357
C07977=1014.464,370.215,343.320,171.535,51.765,160.356
C07978=1014.455,369.968,343.360,171.525,51.767,160.355
C07979=1014.447,369.721,343.398,171.515,51.771,160.354
C07980=1014.440,369.475,343.438,171.506,51.774,160.353
C07981=1014.432,369.227,343.477,171.497,51.777,160.352
C07982=1014.424,368.980,343.517,171.487,51.780,160.351
C07983=1014.415,368.680,343.564,171.476,51.784,160.350
C07984=1014.405,368.378,343.611,171.465,51.787,160.349
C07985=1014.396,368.077,343.659,171.453,51.791,160.347
C07986=1014.386,367.776,343.707,171.442,51.795,160.346
C07987=1014.378,367.530,343.746,171.433,51.798,160.345
C07988=1014.371,367.283,343.785,171.424,51.801,160.344
C07989=1014.362,367.035,343.823,171.415,51.804,160.343
C07990=1014.355,366.789,343.862,171.405,51.808,160.342
C07991=1014.346,366.542,343.901,171.396,51.811,160.341
C07992=1014.339,366.296,343.939,171.387,51.815,160.341
C07993=1014.331,366.049,343.978,171.377,51.817,160.340
C07994=1014.323,365.801,344.016,171.368,51.821,160.339
C07995=1014.315,365.555,344.055,171.359,51.824,160.338
C07996=1014.307,365.308,344.093,171.350,51.828,160.337
C07997=1014.299,365.061,344.131,171.341,51.831,160.336
C07998=1014.291,364.814,344.170,171.332,51.834,160.335
C07999=1014.284,364.567,344.209,171.323,51.837,160.334
C08000=1014.276,364.320,344.248,171.314,51.841,160.333
C08001=1014.269,364.073,344.285,171.305,51.844,160.333
C08002=1014.261,363.826,344.323,171.296,51.848,160.332
C08003=1014.253,363.579,344.362,171.287,51.851,160.331
C08004=1014.246,363.332,344.400,171.278,51.854,160.330
C08005=1014.238,363.085,344.439,171.269,51.858,160.329
C08006=1014.230,362.838,344.476,171.260,51.861,160.328
C08007=1014.223,362.592,344.515,171.251,51.865,160.327
C08008=1014.215,362.344,344.553,171.242,51.868,160.327
C08009=1014.207,362.097,344.591,171.233,51.872,160.326
C08010=1014.200,361.851,344.629,171.224,51.875,160.325
C08011=1014.192,361.603,344.667,171.215,51.878,160.324
C08012=1014.184,361.356,344.705,171.208,51.882,160.324
C08013=1014.177,361.110,344.743,171.199,51.885,160.323
C08014=1014.170,360.863,344.781,171.190,51.889,160.322
C08015=1014.161,360.615,344.819,171.181,51.892,160.321
C08016=1014.154,360.368,344.857,171.172,51.896,160.320
C08017=1014.147,360.121,344.894,171.163,51.900,160.319
C08018=1014.139,359.875,344.933,171.154,51.903,160.319
C08019=1014.132,359.628,344.970,171.145,51.907,160.318
C08020=1014.125,359.381,345.008,171.137,51.911,160.317
C08021=1014.117,359.134,345.046,171.129,51.914,160.316
C08022=1014.110,358.886,345.084,171.120,51.917,160.316
C08023=1014.102,358.640,345.122,171.111,51.921,160.315
C08024=1014.095,358.392,345.160,171.102,51.925,160.314
C08025=1014.088,358.145,345.197,171.094,51.929,160.313
C08026=1014.080,357.898,345.235,171.085,51.932,160.313
C08027=1014.073,357.651,345.272,171.076,51.936,160.312
C08028=1014.065,357.404,345.309,171.068,51.939,160.311
C08029=1014.058,357.157,345.347,171.060,51.943,160.311
C08030=1014.051,356.910,345.384,171.051,51.947,160.310
C08031=1014.043,356.663,345.422,171.042,51.951,160.309
C08032=1014.035,356.416,345.459,171.034,51.955,160.308
C08033=1014.028,356.169,345.496,171.025,51.958,160.308
C08034=1014.021,355.922,345.534,171.017,51.962,160.307
C08035=1014.014,355.674,345.571,171.009,51.966,160.306
C08036=1014.006,355.427,345.608,171.000,51.969,160.305
C08037=1013.999,355.180,345.645,170.991,51.973,160.305
C08038=1013.991,354.933,345.683,170.982,51.977,160.304
C08039=1013.984,354.685,345.719,170.975,51.981,160.304
C08040=1013.977,354.439,345.756,170.966,51.985,160.303
C08041=1013.970,354.192,345.793,170.957,51.989,160.302
C08042=1013.963,353.944,345.830,170.949,51.993,160.302
C08043=1013.954,353.651,345.874,170.939,51.997,160.301
C08044=1013.946,353.357,345.918,170.929,52.002,160.300
C08045=1013.936,353.063,345.962,170.919,52.006,160.299
C08046=1013.928,352.770,346.006,170.910,52.011,160.298
C08047=1013.921,352.523,346.042,170.901,52.015,160.298
C08048=1013.913,352.276,346.079,170.893,52.020,160.297
C08049=1013.906,352.029,346.116,170.884,52.024,160.297
C08050=1013.898,351.782,346.153,170.877,52.027,160.296
C08051=1013.892,351.535,346.190,170.868,52.031,160.296
C08052=1013.884,351.287,346.226,170.860,52.035,160.295
C08053=1013.877,351.040,346.263,170.851,52.040,160.294
C08054=1013.869,350.793,346.299,170.843,52.043,160.294
C08055=1013.863,350.546,346.336,170.835,52.047,160.293
C08056=1013.855,350.298,346.372,170.826,52.051,160.292
C08057=1013.849,350.051,346.409,170.818,52.056,160.292
C08058=1013.841,349.804,346.446,170.811,52.060,160.292
C08059=1013.834,349.557,346.482,170.802,52.064,160.291
C08060=1013.827,349.310,346.518,170.794,52.068,160.290
C08061=1013.820,349.062,346.555,170.786,52.072,160.290
C08062=1013.814,348.815,346.591,170.778,52.076,160.289
C08063=1013.806,348.568,346.628,170.769,52.080,160.289
C08064=1013.800,348.321,346.664,170.762,52.084,160.288
C08065=1013.792,348.073,346.700,170.754,52.089,160.288
C08066=1013.785,347.825,346.737,170.745,52.093,160.287
C08067=1013.778,347.579,346.773,170.738,52.097,160.287
C08068=1013.772,347.332,346.809,170.729,52.101,160.286
C08069=1013.764,347.084,346.846,170.721,52.105,160.285
C08070=1013.757,346.837,346.881,170.714,52.110,160.285
C08071=1013.750,346.589,346.918,170.705,52.114,160.284
C08072=1013.743,346.342,346.953,170.697,52.118,160.284
C08073=1013.736,346.094,346.990,170.689,52.122,160.283
C08074=1013.729,345.848,347.026,170.681,52.127,160.283
C08075=1013.723,345.600,347.061,170.673,52.132,160.283
C08076=1013.715,345.353,347.097,170.666,52.135,160.282
C08077=1013.709,345.106,347.134,170.657,52.140,160.282
C08078=1013.701,344.858,347.169,170.649,52.144,160.281
C08079=1013.694,344.611,347.205,170.642,52.148,160.281
C08080=1013.688,344.363,347.241,170.634,52.153,160.280
C08081=1013.680,344.116,347.277,170.625,52.158,160.280
C08082=1013.674,343.869,347.312,170.618,52.161,160.279
C08083=1013.667,343.622,347.348,170.610,52.166,160.279
C08084=1013.661,343.374,347.384,170.602,52.171,160.278
C08085=1013.653,343.127,347.420,170.595,52.175,160.278
C08086=1013.646,342.879,347.455,170.586,52.179,160.277
C08087=1013.639,342.632,347.490,170.579,52.184,160.277
C08088=1013.633,342.385,347.527,170.571,52.188,160.277
C08089=1013.626,342.137,347.562,170.563,52.193,160.276
C08090=1013.619,341.890,347.597,170.555,52.197,160.276
C08091=1013.612,341.643,347.633,170.547,52.202,160.275
C08092=1013.605,341.395,347.668,170.540,52.207,160.275
C08093=1013.599,341.148,347.704,170.532,52.211,160.274
C08094=1013.592,340.900,347.740,170.523,52.215,160.274
C08095=1013.585,340.652,347.775,170.516,52.220,160.274
C08096=1013.578,340.406,347.811,170.508,52.224,160.273
C08097=1013.571,340.158,347.846,170.501,52.229,160.273
C08098=1013.565,339.911,347.882,170.493,52.233,160.272
C08099=1013.558,339.663,347.917,170.486,52.238,160.272
C08100=1013.551,339.416,347.952,170.478,52.243,160.272
C08101=1013.545,339.168,347.987,170.470,52.248,160.271
C08102=1013.538,338.921,348.022,170.463,52.252,160.271
C08103=1013.530,338.625,348.065,170.454,52.257,160.270
C08104=1013.522,338.329,348.106,170.444,52.264,160.270
C08105=1013.514,338.032,348.148,170.435,52.269,160.270
C08106=1013.506,337.737,348.190,170.426,52.274,160.269
C08107=1013.499,337.489,348.225,170.418,52.279,160.269
C08108=1013.492,337.241,348.260,170.411,52.284,160.269
C08109=1013.486,336.994,348.295,170.403,52.289,160.268
C08110=1013.479,336.747,348.330,170.396,52.293,160.268
C08111=1013.472,336.499,348.364,170.388,52.299,160.268
C08112=1013.466,336.251,348.399,170.380,52.303,160.267
C08113=1013.459,336.004,348.435,170.373,52.308,160.267
C08114=1013.452,335.756,348.469,170.365,52.313,160.267
C08115=1013.445,335.510,348.503,170.358,52.317,160.266
C08116=1013.439,335.262,348.538,170.350,52.322,160.266
C08117=1013.432,335.014,348.573,170.343,52.327,160.266
C08118=1013.425,334.767,348.608,170.335,52.332,160.265
C08119=1013.419,334.519,348.642,170.329,52.337,160.265
C08120=1013.412,334.271,348.677,170.321,52.342,160.265
C08121=1013.406,334.024,348.712,170.314,52.347,160.265
C08122=1013.400,333.777,348.747,170.306,52.351,160.264
C08123=1013.393,333.529,348.781,170.299,52.356,160.264
C08124=1013.387,333.281,348.815,170.291,52.361,160.264
C08125=1013.380,333.034,348.850,170.283,52.367,160.263
C08126=1013.374,332.786,348.885,170.276,52.371,160.263
C08127=1013.366,332.539,348.919,170.268,52.376,160.263
C08128=1013.360,332.291,348.954,170.262,52.381,160.263
C08129=1013.354,332.044,348.988,170.254,52.386,160.262
C08130=1013.347,331.797,349.023,170.247,52.391,160.262
C08131=1013.341,331.549,349.057,170.239,52.397,160.262
C08132=1013.334,331.302,349.091,170.232,52.401,160.262
C08133=1013.328,331.054,349.125,170.224,52.406,160.261
C08134=1013.321,330.806,349.160,170.218,52.411,160.261
C08135=1013.315,330.559,349.193,170.210,52.417,160.261
C08136=1013.308,330.311,349.227,170.203,52.422,160.261
C08137=1013.302,330.063,349.262,170.195,52.427,160.260
C08138=1013.295,329.816,349.295,170.188,52.432,160.260
C08139=1013.289,329.568,349.330,170.181,52.437,160.260
C08140=1013.283,329.320,349.364,170.174,52.442,160.260
C08141=1013.276,329.073,349.398,170.166,52.447,160.260
C08142=1013.270,328.825,349.432,170.160,52.452,160.260
C08143=1013.263,328.577,349.466,170.152,52.458,160.259
C08144=1013.256,328.330,349.500,170.145,52.463,160.259
C08145=1013.250,328.083,349.534,170.138,52.468,160.259
C08146=1013.243,327.835,349.568,170.130,52.473,160.259
C08147=1013.238,327.587,349.601,170.123,52.478,160.258
C08148=1013.232,327.340,349.635,170.116,52.483,160.258
C08149=1013.225,327.092,349.669,170.108,52.488,160.258
C08150=1013.219,326.845,349.703,170.102,52.494,160.258
C08151=1013.212,326.597,349.737,170.094,52.500,160.258
C08152=1013.206,326.349,349.770,170.088,52.505,160.258
C08153=1013.199,326.101,349.805,170.080,52.510,160.257
C08154=1013.194,325.854,349.839,170.073,52.515,160.257
C08155=1013.187,325.606,349.871,170.067,52.520,160.257
C08156=1013.180,325.359,349.905,170.059,52.526,160.257
C08157=1013.175,325.111,349.939,170.051,52.531,160.257
C08158=1013.168,324.864,349.972,170.045,52.537,160.257
C08159=1013.161,324.615,350.005,170.037,52.542,160.257
C08160=1013.154,324.368,350.039,170.031,52.547,160.256
C08161=1013.148,324.121,350.071,170.023,52.553,160.256
C08162=1013.142,323.872,350.105,170.017,52.558,160.256
C08163=1013.134,323.572,350.145,170.008,52.565,160.256
C08164=1013.126,323.272,350.186,169.999,52.572,160.256
C08165=1013.118,322.971,350.226,169.991,52.578,160.256
C08166=1013.111,322.671,350.266,169.983,52.584,160.256
C08167=1013.104,322.423,350.299,169.975,52.591,160.256
C08168=1013.098,322.176,350.332,169.969,52.596,160.256
C08169=1013.091,321.927,350.365,169.961,52.601,160.255
C08170=1013.085,321.680,350.399,169.955,52.607,160.255
C08171=1013.079,321.432,350.432,169.947,52.612,160.255
C08172=1013.073,321.185,350.464,169.941,52.618,160.255
C08173=1013.066,320.937,350.497,169.933,52.623,160.255
C08174=1013.060,320.689,350.530,169.927,52.629,160.255
C08175=1013.053,320.441,350.563,169.919,52.634,160.255
C08176=1013.048,320.193,350.596,169.913,52.640,160.255
C08177=1013.041,319.946,350.629,169.906,52.646,160.255
C08178=1013.035,319.698,350.662,169.899,52.651,160.255
C08179=1013.029,319.451,350.694,169.892,52.657,160.255
C08180=1013.023,319.203,350.727,169.885,52.663,160.255
C08181=1013.017,318.955,350.761,169.878,52.669,160.255
C08182=1013.010,318.707,350.794,169.872,52.674,160.255
C08183=1013.004,318.459,350.826,169.864,52.680,160.255
C08184=1012.998,318.212,350.859,169.858,52.685,160.255
C08185=1012.991,317.964,350.892,169.850,52.692,160.255
C08186=1012.986,317.716,350.925,169.844,52.697,160.254
C08187=1012.979,317.469,350.958,169.837,52.703,160.254
C08188=1012.973,317.220,350.990,169.830,52.708,160.255
C08189=1012.967,316.973,351.023,169.824,52.714,160.255
C08190=1012.961,316.725,351.055,169.816,52.720,160.254
C08191=1012.955,316.478,351.088,169.810,52.725,160.254
C08192=1012.949,316.230,351.122,169.803,52.731,160.254
C08193=1012.944,315.982,351.153,169.797,52.737,160.255
C08194=1012.937,315.735,351.186,169.789,52.743,160.254
C08195=1012.931,315.487,351.219,169.783,52.748,160.254
C08196=1012.925,315.239,351.251,169.775,52.755,160.254
C08197=1012.919,314.991,351.284,169.769,52.760,160.254
C08198=1012.913,314.743,351.317,169.763,52.766,160.254
C08199=1012.907,314.495,351.349,169.756,52.772,160.254
C08200=1012.901,314.247,351.382,169.750,52.778,160.255
C08201=1012.895,314.001,351.414,169.742,52.784,160.254
C08202=1012.889,313.752,351.446,169.736,52.790,160.255
C08203=1012.884,313.504,351.479,169.729,52.796,160.255
C08204=1012.878,313.256,351.511,169.723,52.802,160.255
C08205=1012.871,313.009,351.544,169.715,52.808,160.255
C08206=1012.866,312.761,351.576,169.709,52.813,160.255
C08207=1012.860,312.514,351.608,169.703,52.819,160.255
C08208=1012.854,312.265,351.641,169.696,52.825,160.255
C08209=1012.848,312.017,351.674,169.689,52.831,160.255
C08210=1012.843,311.770,351.706,169.682,52.837,160.255
C08211=1012.836,311.522,351.738,169.676,52.843,160.255
C08212=1012.830,311.274,351.770,169.670,52.849,160.255
C08213=1012.825,311.027,351.803,169.662,52.855,160.255
C08214=1012.819,310.779,351.835,169.656,52.861,160.255
C08215=1012.814,310.530,351.867,169.649,52.867,160.255
C08216=1012.808,310.284,351.900,169.643,52.872,160.255
C08217=1012.802,310.035,351.932,169.637,52.879,160.255
C08218=1012.796,309.787,351.964,169.630,52.885,160.255
C08219=1012.790,309.540,351.996,169.624,52.891,160.255
C08220=1012.784,309.292,352.028,169.616,52.897,160.255
C08221=1012.780,309.044,352.060,169.610,52.903,160.255
C08222=1012.773,308.796,352.092,169.603,52.909,160.256
C08223=1012.766,308.501,352.129,169.595,52.917,160.256
C08224=1012.758,308.207,352.167,169.588,52.924,160.256
C08225=1012.752,307.911,352.205,169.580,52.931,160.256
C08226=1012.744,307.616,352.242,169.573,52.939,160.256
C08227=1012.738,307.369,352.273,169.565,52.945,160.256
C08228=1012.732,307.121,352.305,169.560,52.951,160.256
C08229=1012.726,306.873,352.337,169.552,52.958,160.256
C08230=1012.720,306.625,352.368,169.547,52.964,160.257
C08231=1012.714,306.377,352.399,169.539,52.970,160.257
C08232=1012.708,306.130,352.431,169.534,52.977,160.257
C08233=1012.702,305.882,352.462,169.526,52.983,160.257
C08234=1012.697,305.634,352.493,169.521,52.989,160.257
C08235=1012.690,305.386,352.525,169.514,52.995,160.257
C08236=1012.684,305.138,352.556,169.508,53.002,160.257
C08237=1012.678,304.890,352.587,169.501,53.008,160.258
C08238=1012.673,304.642,352.619,169.495,53.014,160.258
C08239=1012.666,304.394,352.650,169.489,53.021,160.258
C08240=1012.661,304.146,352.681,169.482,53.027,160.258
C08241=1012.655,303.899,352.712,169.476,53.033,160.258
C08242=1012.649,303.650,352.743,169.469,53.040,160.258
C08243=1012.643,303.403,352.774,169.463,53.046,160.259
C08244=1012.637,303.154,352.806,169.456,53.053,160.259
C08245=1012.631,302.907,352.837,169.450,53.059,160.259
C08246=1012.626,302.659,352.868,169.443,53.065,160.259
C08247=1012.620,302.410,352.900,169.437,53.072,160.259
C08248=1012.614,302.163,352.930,169.431,53.079,160.259
C08249=1012.608,301.914,352.962,169.425,53.085,160.260
C08250=1012.602,301.667,352.993,169.418,53.092,160.260
C08251=1012.597,301.419,353.024,169.412,53.098,160.260
C08252=1012.591,301.171,353.055,169.405,53.105,160.260
C08253=1012.586,300.922,353.086,169.399,53.111,160.260
C08254=1012.579,300.675,353.117,169.392,53.118,160.261
C08255=1012.574,300.427,353.148,169.387,53.124,160.261
C08256=1012.568,300.179,353.179,169.379,53.131,160.261
C08257=1012.563,299.931,353.210,169.374,53.137,160.261
C08258=1012.557,299.683,353.241,169.367,53.144,160.261
C08259=1012.552,299.435,353.272,169.361,53.150,160.262
C08260=1012.545,299.187,353.302,169.354,53.157,160.262
C08261=1012.540,298.939,353.334,169.349,53.164,160.262
C08262=1012.534,298.691,353.364,169.343,53.170,160.262
C08263=1012.529,298.443,353.395,169.336,53.177,160.263
C08264=1012.523,298.195,353.426,169.330,53.183,160.263
C08265=1012.517,297.947,353.458,169.324,53.190,160.263
C08266=1012.511,297.699,353.488,169.318,53.197,160.263
C08267=1012.506,297.451,353.519,169.311,53.204,160.264
C08268=1012.500,297.203,353.549,169.305,53.210,160.264
C08269=1012.495,296.955,353.580,169.299,53.217,160.264
C08270=1012.490,296.707,353.611,169.293,53.223,160.264
C08271=1012.484,296.459,353.642,169.286,53.230,160.264
C08272=1012.478,296.211,353.672,169.280,53.237,160.265
C08273=1012.473,295.963,353.703,169.274,53.244,160.265
C08274=1012.467,295.715,353.734,169.268,53.250,160.265
C08275=1012.462,295.467,353.764,169.262,53.257,160.266
C08276=1012.456,295.219,353.795,169.255,53.264,160.266
C08277=1012.451,294.971,353.826,169.250,53.270,160.266
C08278=1012.445,294.723,353.856,169.243,53.278,160.266
C08279=1012.440,294.475,353.887,169.238,53.284,160.267
C08280=1012.434,294.227,353.917,169.231,53.291,160.267
C08281=1012.429,293.979,353.948,169.225,53.297,160.267
C08282=1012.424,293.731,353.979,169.218,53.304,160.267
C08283=1012.418,293.454,354.014,169.212,53.312,160.268
C08284=1012.412,293.177,354.047,169.205,53.320,160.268
C08285=1012.406,292.901,354.081,169.198,53.327,160.268
C08286=1012.400,292.624,354.115,169.192,53.335,160.269
C08287=1012.395,292.376,354.146,169.185,53.342,160.269
C08288=1012.389,292.128,354.176,169.180,53.348,160.269
C08289=1012.383,291.880,354.206,169.173,53.356,160.270
C08290=1012.378,291.632,354.236,169.168,53.362,160.270
C08291=1012.373,291.384,354.267,169.161,53.369,160.270
C08292=1012.367,291.135,354.297,169.156,53.376,160.271
C08293=1012.361,290.887,354.327,169.149,53.383,160.271
C08294=1012.356,290.639,354.357,169.144,53.390,160.271
C08295=1012.350,290.391,354.387,169.137,53.397,160.271
C08296=1012.345,290.143,354.416,169.132,53.405,160.272
C08297=1012.339,289.895,354.447,169.125,53.411,160.272
C08298=1012.334,289.647,354.476,169.119,53.419,160.273
C08299=1012.328,289.399,354.506,169.113,53.426,160.273
C08300=1012.322,289.151,354.536,169.107,53.433,160.273
C08301=1012.317,288.902,354.566,169.101,53.440,160.274
C08302=1012.311,288.655,354.596,169.095,53.447,160.274
C08303=1012.306,288.407,354.625,169.089,53.454,160.274
C08304=1012.301,288.158,354.656,169.083,53.461,160.275
C08305=1012.296,287.910,354.685,169.077,53.468,160.275
C08306=1012.290,287.662,354.716,169.070,53.475,160.275
C08307=1012.284,287.413,354.745,169.065,53.483,160.276
C08308=1012.280,287.166,354.775,169.059,53.490,160.276
C08309=1012.274,286.917,354.804,169.053,53.497,160.276
C08310=1012.268,286.669,354.835,169.047,53.504,160.277
C08311=1012.263,286.421,354.864,169.041,53.512,160.277
C08312=1012.258,286.173,354.894,169.035,53.518,160.278
C08313=1012.252,285.925,354.923,169.029,53.526,160.278
C08314=1012.246,285.677,354.952,169.023,53.533,160.278
C08315=1012.241,285.429,354.981,169.017,53.540,160.279
C08316=1012.236,285.180,355.011,169.011,53.547,160.279
C08317=1012.230,284.932,355.041,169.005,53.555,160.280
C08318=1012.224,284.684,355.071,169.000,53.562,160.280
C08319=1012.219,284.436,355.100,168.994,53.570,160.280
C08320=1012.214,284.188,355.130,168.988,53.576,160.281
C08321=1012.208,283.939,355.160,168.982,53.584,160.281
C08322=1012.203,283.692,355.189,168.975,53.591,160.281
C08323=1012.198,283.443,355.217,168.970,53.599,160.282
C08324=1012.192,283.195,355.247,168.964,53.606,160.282
C08325=1012.187,282.947,355.276,168.959,53.613,160.283
C08326=1012.181,282.699,355.305,168.952,53.621,160.283
C08327=1012.176,282.451,355.334,168.946,53.629,160.284
C08328=1012.171,282.202,355.363,168.941,53.636,160.284
C08329=1012.165,281.953,355.393,168.935,53.644,160.285
C08330=1012.160,281.706,355.422,168.929,53.651,160.285
C08331=1012.151,281.335,355.465,168.920,53.661,160.285
C08332=1012.143,280.964,355.509,168.911,53.673,160.286
C08333=1012.135,280.594,355.552,168.902,53.684,160.287
C08334=1012.127,280.222,355.595,168.893,53.695,160.287
C08335=1011.905,282.016,355.022,168.907,53.731,160.298
C08336=1011.909,282.229,354.997,168.911,53.724,160.298
C08337=1011.914,282.440,354.971,168.916,53.718,160.297
C08338=1011.919,282.652,354.947,168.922,53.711,160.297
C08339=1011.923,282.864,354.922,168.927,53.705,160.297
C08340=1011.928,283.076,354.897,168.931,53.699,160.296
C08341=1011.933,283.289,354.872,168.937,53.692,160.296
C08342=1011.937,283.501,354.847,168.942,53.686,160.296
C08343=1011.942,283.712,354.822,168.947,53.679,160.295
C08344=1011.947,283.960,354.793,168.953,53.672,160.295
C08345=1011.953,284.209,354.763,168.959,53.665,160.295
C08346=1011.958,284.457,354.734,168.965,53.658,160.294
C08347=1011.963,284.705,354.704,168.971,53.650,160.294
C08348=1011.969,284.953,354.675,168.976,53.643,160.293
C08349=1011.974,285.201,354.646,168.982,53.636,160.293
C08350=1011.980,285.449,354.616,168.989,53.629,160.293
C08351=1011.985,285.698,354.587,168.994,53.621,160.292
C08352=1011.990,285.946,354.557,169.001,53.614,160.292
C08353=1011.996,286.194,354.528,169.006,53.607,160.291
C08354=1012.001,286.442,354.498,169.013,53.600,160.291
C08355=1012.006,286.690,354.469,169.019,53.592,160.291
C08356=1012.012,286.939,354.439,169.024,53.585,160.290
C08357=1012.017,287.187,354.409,169.031,53.578,160.290
C08358=1012.022,287.434,354.379,169.036,53.571,160.290
C08359=1012.028,287.683,354.350,169.042,53.563,160.289
C08360=1012.033,287.931,354.320,169.048,53.557,160.289
C08361=1012.039,288.180,354.291,169.054,53.549,160.289
C08362=1012.045,288.427,354.260,169.060,53.542,160.288
C08363=1012.050,288.675,354.231,169.066,53.535,160.288
C08364=1012.055,288.924,354.201,169.073,53.528,160.288
C08365=1012.061,289.172,354.172,169.078,53.521,160.287
C08366=1012.066,289.420,354.141,169.085,53.513,160.287
C08367=1012.072,289.668,354.112,169.090,53.507,160.287
C08368=1012.077,289.916,354.082,169.096,53.499,160.286
C08369=1012.083,290.164,354.052,169.102,53.492,160.286
C08370=1012.088,290.412,354.022,169.108,53.485,160.286
C08371=1012.093,290.660,353.991,169.115,53.478,160.285
C08372=1012.099,290.909,353.962,169.121,53.471,160.285
C08373=1012.105,291.157,353.931,169.127,53.464,160.285
C08374=1012.110,291.405,353.902,169.133,53.457,160.284
C08375=1012.116,291.653,353.871,169.139,53.450,160.284
C08376=1012.121,291.901,353.842,169.145,53.443,160.284
C08377=1012.127,292.148,353.812,169.152,53.436,160.284
C08378=1012.132,292.397,353.781,169.157,53.429,160.283
C08379=1012.137,292.645,353.751,169.164,53.422,160.283
C08380=1012.144,292.924,353.716,169.170,53.415,160.282
C08381=1012.149,293.202,353.683,169.177,53.407,160.282
C08382=1012.155,293.482,353.648,169.184,53.399,160.282
C08383=1012.161,293.761,353.614,169.191,53.391,160.281
C08384=1012.166,294.009,353.583,169.198,53.384,160.281
C08385=1012.172,294.257,353.553,169.203,53.378,160.281
C08386=1012.177,294.505,353.522,169.210,53.371,160.281
C08387=1012.182,294.753,353.491,169.216,53.364,160.281
C08388=1012.188,295.001,353.461,169.223,53.358,160.280
C08389=1012.193,295.249,353.430,169.228,53.350,160.280
C08390=1012.199,295.497,353.400,169.234,53.344,160.280
C08391=1012.204,295.745,353.369,169.240,53.337,160.279
C08392=1012.210,295.993,353.338,169.246,53.331,160.279
C08393=1012.215,296.241,353.307,169.253,53.324,160.279
C08394=1012.221,296.489,353.277,169.259,53.317,160.279
C08395=1012.226,296.737,353.246,169.265,53.310,160.279
C08396=1012.232,296.985,353.216,169.271,53.304,160.278
C08397=1012.237,297.233,353.185,169.278,53.297,160.278
C08398=1012.243,297.482,353.154,169.284,53.290,160.278
C08399=1012.248,297.730,353.123,169.290,53.284,160.278
C08400=1012.254,297.978,353.093,169.296,53.277,160.277
C08401=1012.259,298.226,353.062,169.303,53.270,160.277
C08402=1012.265,298.474,353.031,169.309,53.264,160.277
C08403=1012.271,298.721,353.000,169.315,53.257,160.277
C08404=1012.276,298.969,352.969,169.322,53.250,160.277
C08405=1012.282,299.218,352.938,169.328,53.243,160.276
C08406=1012.288,299.466,352.908,169.335,53.237,160.276
C08407=1012.293,299.714,352.877,169.340,53.230,160.276
C08408=1012.299,299.961,352.846,169.347,53.223,160.276
C08409=1012.304,300.209,352.815,169.353,53.217,160.275
C08410=1012.311,300.458,352.784,169.360,53.210,160.275
C08411=1012.316,300.706,352.753,169.366,53.204,160.275
C08412=1012.322,300.953,352.722,169.373,53.197,160.275
C08413=1012.327,301.201,352.691,169.378,53.191,160.275
C08414=1012.333,301.449,352.660,169.385,53.184,160.274
C08415=1012.339,301.697,352.629,169.391,53.177,160.274
C08416=1012.344,301.945,352.598,169.398,53.171,160.274
C08417=1012.350,302.193,352.566,169.404,53.165,160.274
C08418=1012.356,302.441,352.535,169.410,53.158,160.274
C08419=1012.361,302.689,352.505,169.416,53.152,160.273
C08420=1012.367,302.937,352.473,169.423,53.145,160.273
C08421=1012.373,303.185,352.443,169.429,53.139,160.273
C08422=1012.379,303.433,352.411,169.436,53.132,160.273
C08423=1012.385,303.681,352.380,169.442,53.126,160.273
C08424=1012.390,303.929,352.349,169.449,53.119,160.273
C08425=1012.397,304.177,352.318,169.455,53.113,160.272
C08426=1012.402,304.425,352.286,169.461,53.106,160.272
C08427=1012.408,304.672,352.256,169.468,53.100,160.272
C08428=1012.414,304.921,352.224,169.474,53.093,160.272
C08429=1012.420,305.168,352.193,169.481,53.088,160.272
C08430=1012.426,305.417,352.162,169.487,53.081,160.272
C08431=1012.432,305.664,352.130,169.494,53.074,160.272
C08432=1012.438,305.912,352.098,169.500,53.068,160.271
C08433=1012.444,306.160,352.068,169.507,53.061,160.271
C08434=1012.450,306.408,352.036,169.513,53.056,160.271
C08435=1012.456,306.655,352.005,169.520,53.049,160.271
C08436=1012.461,306.904,351.974,169.526,53.043,160.271
C08437=1012.468,307.151,351.943,169.533,53.036,160.271
C08438=1012.474,307.400,351.911,169.539,53.030,160.271
C08439=1012.480,307.647,351.880,169.546,53.024,160.271
C08440=1012.487,307.945,351.842,169.554,53.016,160.270
C08441=1012.494,308.242,351.804,169.561,53.008,160.270
C08442=1012.501,308.538,351.766,169.570,53.001,160.270
C08443=1012.509,308.836,351.728,169.578,52.994,160.270
C08444=1012.515,309.084,351.696,169.584,52.988,160.270
C08445=1012.520,309.331,351.665,169.591,52.981,160.270
C08446=1012.526,309.580,351.633,169.597,52.975,160.270
C08447=1012.531,309.828,351.600,169.604,52.969,160.270
C08448=1012.537,310.075,351.568,169.610,52.963,160.270
C08449=1012.542,310.323,351.536,169.618,52.957,160.270
C08450=1012.548,310.571,351.504,169.623,52.951,160.269
C08451=1012.555,310.818,351.471,169.630,52.945,160.269
C08452=1012.560,311.066,351.440,169.637,52.939,160.269
C08453=1012.566,311.314,351.407,169.643,52.933,160.269
C08454=1012.571,311.562,351.374,169.650,52.927,160.269
C08455=1012.577,311.810,351.343,169.657,52.921,160.269
C08456=1012.583,312.058,351.310,169.664,52.915,160.269
C08457=1012.589,312.305,351.278,169.670,52.909,160.269
C08458=1012.595,312.553,351.246,169.677,52.903,160.269
C08459=1012.601,312.800,351.213,169.684,52.897,160.269
C08460=1012.606,313.049,351.181,169.690,52.891,160.269
C08461=1012.612,313.297,351.148,169.697,52.885,160.269
C08462=1012.618,313.544,351.116,169.704,52.879,160.269
C08463=1012.624,313.792,351.084,169.710,52.873,160.269
C08464=1012.630,314.040,351.052,169.717,52.868,160.269
C08465=1012.636,314.288,351.018,169.724,52.862,160.269
C08466=1012.641,314.535,350.987,169.730,52.856,160.269
C08467=1012.647,314.783,350.954,169.737,52.850,160.269
C08468=1012.654,315.030,350.921,169.744,52.844,160.269
C08469=1012.660,315.279,350.889,169.751,52.838,160.269
C08470=1012.666,315.526,350.856,169.757,52.832,160.269
C08471=1012.671,315.774,350.823,169.764,52.826,160.269
C08472=1012.677,316.022,350.791,169.770,52.820,160.269
C08473=1012.683,316.269,350.759,169.778,52.814,160.269
C08474=1012.689,316.517,350.726,169.784,52.809,160.269
C08475=1012.695,316.765,350.694,169.792,52.803,160.269
C08476=1012.702,317.013,350.661,169.798,52.797,160.269
C08477=1012.707,317.261,350.628,169.805,52.791,160.269
C08478=1012.713,317.508,350.595,169.812,52.786,160.269
C08479=1012.719,317.756,350.563,169.819,52.780,160.269
C08480=1012.726,318.004,350.530,169.825,52.774,160.269
C08481=1012.732,318.252,350.497,169.832,52.768,160.269
C08482=1012.738,318.500,350.464,169.839,52.763,160.269
C08483=1012.744,318.747,350.431,169.846,52.757,160.269
C08484=1012.750,318.995,350.399,169.853,52.751,160.269
C08485=1012.756,319.242,350.366,169.860,52.746,160.269
C08486=1012.763,319.490,350.333,169.867,52.740,160.269
C08487=1012.769,319.737,350.300,169.874,52.734,160.269
C08488=1012.775,319.986,350.267,169.881,52.728,160.270
C08489=1012.782,320.234,350.234,169.888,52.723,160.270
C08490=1012.788,320.481,350.201,169.895,52.717,160.270
C08491=1012.794,320.729,350.168,169.902,52.712,160.270
C08492=1012.800,320.976,350.136,169.909,52.705,160.270
C08493=1012.806,321.224,350.102,169.916,52.700,160.270
C08494=1012.812,321.472,350.070,169.923,52.694,160.270
C08495=1012.819,321.720,350.037,169.929,52.689,160.270
C08496=1012.825,321.968,350.004,169.937,52.683,160.270
C08497=1012.832,322.215,349.971,169.943,52.678,160.270
C08498=1012.837,322.463,349.938,169.951,52.672,160.270
C08499=1012.844,322.711,349.905,169.957,52.667,160.270
C08500=1012.851,323.013,349.864,169.967,52.660,160.271
C08501=1012.859,323.316,349.824,169.975,52.654,160.271
C08502=1012.868,323.618,349.783,169.984,52.646,160.271
C08503=1012.875,323.921,349.743,169.992,52.640,160.271
C08504=1012.883,324.169,349.709,170.000,52.634,160.271
C08505=1012.888,324.417,349.676,170.006,52.629,160.271
C08506=1012.894,324.665,349.643,170.013,52.623,160.271
C08507=1012.901,324.913,349.610,170.021,52.618,160.271
C08508=1012.908,325.160,349.577,170.028,52.612,160.272
C08509=1012.914,325.407,349.544,170.035,52.606,160.272
C08510=1012.921,325.655,349.509,170.042,52.601,160.272
C08511=1012.927,325.903,349.477,170.049,52.596,160.272
C08512=1012.933,326.150,349.443,170.056,52.591,160.272
C08513=1012.939,326.398,349.408,170.064,52.585,160.272
C08514=1012.946,326.645,349.375,170.071,52.580,160.272
C08515=1012.951,326.893,349.341,170.078,52.575,160.273
C08516=1012.958,327.141,349.307,170.085,52.570,160.273
C08517=1012.964,327.388,349.274,170.093,52.564,160.273
C08518=1012.971,327.636,349.239,170.099,52.559,160.273
C08519=1012.977,327.884,349.206,170.107,52.554,160.273
C08520=1012.984,328.132,349.172,170.115,52.549,160.274
C08521=1012.990,328.379,349.138,170.121,52.544,160.274
C08522=1012.997,328.627,349.104,170.129,52.538,160.274
C08523=1013.003,328.874,349.070,170.136,52.533,160.274
C08524=1013.009,329.122,349.036,170.143,52.528,160.274
C08525=1013.015,329.370,349.003,170.150,52.523,160.274
C08526=1013.022,329.618,348.968,170.158,52.517,160.275
C08527=1013.028,329.865,348.934,170.164,52.512,160.275
C08528=1013.035,330.112,348.901,170.172,52.507,160.275
C08529=1013.041,330.360,348.867,170.180,52.501,160.275
C08530=1013.047,330.608,348.832,170.186,52.496,160.275
C08531=1013.054,330.855,348.798,170.195,52.492,160.276
C08532=1013.060,331.103,348.764,170.201,52.486,160.276
C08533=1013.067,331.351,348.730,170.209,52.481,160.276
C08534=1013.074,331.598,348.695,170.216,52.476,160.276
C08535=1013.080,331.845,348.661,170.223,52.471,160.277
C08536=1013.087,332.093,348.627,170.232,52.466,160.277
C08537=1013.093,332.341,348.592,170.238,52.461,160.277
C08538=1013.099,332.588,348.558,170.246,52.455,160.277
C08539=1013.106,332.836,348.523,170.253,52.451,160.278
C08540=1013.113,333.083,348.489,170.261,52.446,160.278
C08541=1013.119,333.330,348.455,170.268,52.441,160.278
C08542=1013.126,333.578,348.420,170.276,52.436,160.279
C08543=1013.132,333.826,348.386,170.283,52.430,160.279
C08544=1013.139,334.073,348.351,170.290,52.426,160.279
C08545=1013.145,334.321,348.317,170.298,52.421,160.279
C08546=1013.151,334.568,348.281,170.305,52.416,160.280
C08547=1013.158,334.816,348.247,170.313,52.411,160.280
C08548=1013.165,335.063,348.212,170.320,52.407,160.280
C08549=1013.171,335.311,348.177,170.328,52.401,160.281
C08550=1013.177,335.558,348.143,170.336,52.396,160.281
C08551=1013.184,335.806,348.109,170.342,52.391,160.281
C08552=1013.191,336.053,348.074,170.351,52.387,160.282
C08553=1013.198,336.301,348.039,170.358,52.382,160.282
C08554=1013.204,336.548,348.004,170.365,52.377,160.282
C08555=1013.211,336.796,347.969,170.374,52.372,160.283
C08556=1013.218,337.044,347.935,170.381,52.368,160.283
C08557=1013.224,337.291,347.899,170.388,52.362,160.283
C08558=1013.231,337.538,347.864,170.397,52.358,160.284
C08559=1013.238,337.786,347.829,170.404,52.353,160.284
C08560=1013.246,338.084,347.788,170.413,52.347,160.284
C08561=1013.254,338.383,347.746,170.422,52.341,160.285
C08562=1013.262,338.681,347.703,170.431,52.335,160.285
C08563=1013.270,338.979,347.661,170.441,52.330,160.286
C08564=1013.276,339.227,347.626,170.448,52.326,160.286
C08565=1013.283,339.474,347.591,170.456,52.321,160.286
C08566=1013.289,339.722,347.555,170.464,52.315,160.287
C08567=1013.296,339.968,347.520,170.471,52.311,160.287
C08568=1013.304,340.216,347.484,170.479,52.306,160.287
C08569=1013.311,340.464,347.449,170.486,52.302,160.288
C08570=1013.317,340.711,347.413,170.494,52.297,160.288
C08571=1013.323,340.959,347.378,170.502,52.293,160.289
C08572=1013.330,341.206,347.343,170.510,52.288,160.289
C08573=1013.337,341.454,347.308,170.518,52.283,160.289
C08574=1013.344,341.701,347.273,170.526,52.279,160.290
C08575=1013.351,341.948,347.237,170.533,52.274,160.290
C08576=1013.357,342.196,347.201,170.541,52.270,160.291
C08577=1013.364,342.443,347.166,170.549,52.265,160.291
C08578=1013.371,342.690,347.130,170.557,52.261,160.292
C08579=1013.378,342.937,347.095,170.565,52.256,160.292
C08580=1013.384,343.185,347.059,170.573,52.252,160.292
C08581=1013.392,343.433,347.023,170.580,52.247,160.293
C08582=1013.399,343.680,346.988,170.588,52.243,160.293
C08583=1013.406,343.927,346.952,170.596,52.238,160.294
C08584=1013.412,344.174,346.916,170.604,52.234,160.294
C08585=1013.419,344.422,346.880,170.612,52.229,160.295
C08586=1013.426,344.669,346.845,170.620,52.225,160.295
C08587=1013.433,344.916,346.809,170.629,52.221,160.296
C08588=1013.440,345.164,346.773,170.636,52.216,160.296
C08589=1013.447,345.411,346.737,170.644,52.212,160.297
C08590=1013.454,345.658,346.702,170.652,52.207,160.297
C08591=1013.461,345.906,346.665,170.660,52.203,160.298
C08592=1013.467,346.154,346.630,170.668,52.198,160.298
C08593=1013.475,346.401,346.594,170.676,52.194,160.299
C08594=1013.481,346.648,346.557,170.685,52.190,160.299
C08595=1013.488,346.895,346.521,170.692,52.186,160.300
C08596=1013.495,347.143,346.484,170.700,52.181,160.300
C08597=1013.502,347.390,346.449,170.709,52.177,160.301
C08598=1013.510,347.637,346.413,170.716,52.173,160.301
C08599=1013.516,347.884,346.377,170.724,52.169,160.302
C08600=1013.523,348.132,346.340,170.733,52.164,160.302
C08601=1013.530,348.379,346.304,170.741,52.160,160.303
C08602=1013.537,348.627,346.267,170.748,52.155,160.303
C08603=1013.544,348.873,346.231,170.757,52.151,160.304
C08604=1013.551,349.121,346.195,170.765,52.147,160.304
C08605=1013.558,349.368,346.159,170.774,52.143,160.305
C08606=1013.565,349.616,346.122,170.781,52.139,160.305
C08607=1013.572,349.862,346.086,170.790,52.135,160.306
C08608=1013.579,350.110,346.048,170.798,52.131,160.307
C08609=1013.587,350.357,346.012,170.806,52.126,160.307
C08610=1013.593,350.604,345.976,170.814,52.122,160.308
C08611=1013.601,350.851,345.940,170.822,52.118,160.308
C08612=1013.608,351.099,345.903,170.831,52.114,160.309
C08613=1013.615,351.345,345.866,170.840,52.110,160.310
C08614=1013.622,351.593,345.829,170.848,52.105,160.310
C08615=1013.630,351.841,345.793,170.855,52.102,160.311
C08616=1013.637,352.087,345.756,170.864,52.098,160.311
C08617=1013.644,352.334,345.720,170.872,52.094,160.312
C08618=1013.651,352.582,345.683,170.881,52.089,160.313
C08619=1013.659,352.829,345.646,170.889,52.085,160.313
C08620=1013.667,353.126,345.602,170.899,52.081,160.314
C08621=1013.676,353.420,345.558,170.910,52.076,160.315
C08622=1013.685,353.716,345.514,170.919,52.071,160.315
C08623=1013.693,354.012,345.470,170.929,52.066,160.316
C08624=1013.701,354.259,345.433,170.938,52.062,160.317
C08625=1013.708,354.506,345.395,170.947,52.059,160.318
C08626=1013.715,354.754,345.358,170.954,52.055,160.318
C08627=1013.722,355.000,345.322,170.963,52.051,160.319
C08628=1013.729,355.247,345.284,170.971,52.047,160.319
C08629=1013.736,355.495,345.247,170.980,52.043,160.320
C08630=1013.744,355.742,345.210,170.989,52.039,160.321
C08631=1013.752,355.989,345.173,170.998,52.035,160.322
C08632=1013.759,356.236,345.135,171.006,52.031,160.322
C08633=1013.766,356.483,345.098,171.014,52.028,160.323
C08634=1013.774,356.730,345.061,171.023,52.024,160.324
C08635=1013.781,356.977,345.023,171.031,52.020,160.324
C08636=1013.788,357.225,344.987,171.040,52.016,160.325
C08637=1013.795,357.472,344.949,171.049,52.013,160.326
C08638=1013.803,357.719,344.912,171.057,52.008,160.326
C08639=1013.811,357.966,344.874,171.066,52.004,160.327
C08640=1013.818,358.213,344.836,171.075,52.001,160.328
C08641=1013.826,358.460,344.799,171.083,51.997,160.329
C08642=1013.833,358.707,344.761,171.092,51.993,160.329
C08643=1013.840,358.954,344.724,171.101,51.989,160.330
C08644=1013.847,359.201,344.686,171.109,51.986,160.331
C08645=1013.855,359.448,344.648,171.118,51.983,160.332
C08646=1013.863,359.696,344.610,171.126,51.979,160.332
C08647=1013.870,359.943,344.573,171.135,51.975,160.333
C08648=1013.877,360.189,344.534,171.144,51.972,160.334
C08649=1013.885,360.436,344.497,171.153,51.968,160.335
C08650=1013.892,360.683,344.459,171.162,51.964,160.336
C08651=1013.899,360.930,344.421,171.171,51.961,160.336
C08652=1013.907,361.178,344.383,171.179,51.957,160.337
C08653=1013.915,361.424,344.345,171.188,51.954,160.338
C08654=1013.922,361.672,344.307,171.197,51.950,160.339
C08655=1013.930,361.918,344.269,171.206,51.947,160.340
C08656=1013.938,362.165,344.231,171.215,51.943,160.340
C08657=1013.945,362.412,344.193,171.224,51.939,160.341
C08658=1013.953,362.659,344.155,171.233,51.936,160.342
C08659=1013.961,362.906,344.116,171.242,51.932,160.343
C08660=1013.968,363.153,344.079,171.251,51.929,160.344
C08661=1013.976,363.400,344.040,171.260,51.925,160.344
C08662=1013.984,363.647,344.002,171.269,51.922,160.345
C08663=1013.991,363.894,343.964,171.278,51.919,160.346
C08664=1013.999,364.141,343.926,171.287,51.915,160.347
C08665=1014.006,364.388,343.887,171.296,51.912,160.348
C08666=1014.013,364.635,343.849,171.305,51.908,160.349
C08667=1014.022,364.882,343.810,171.314,51.905,160.350
C08668=1014.029,365.128,343.772,171.323,51.901,160.350
C08669=1014.037,365.376,343.733,171.332,51.898,160.351
C08670=1014.045,365.622,343.695,171.342,51.894,160.352
C08671=1014.053,365.869,343.656,171.351,51.891,160.353
C08672=1014.061,366.116,343.618,171.360,51.888,160.354
C08673=1014.069,366.363,343.579,171.369,51.885,160.355
C08674=1014.077,366.610,343.541,171.378,51.881,160.356
C08675=1014.084,366.857,343.503,171.387,51.878,160.357
C08676=1014.093,367.104,343.464,171.396,51.875,160.358
C08677=1014.099,367.351,343.425,171.405,51.872,160.359
C08678=1014.108,367.597,343.386,171.416,51.868,160.360
C08679=1014.115,367.844,343.348,171.425,51.865,160.361
C08680=1014.126,368.148,343.299,171.436,51.861,160.362
C08681=1014.135,368.451,343.251,171.447,51.857,160.363
C08682=1014.144,368.754,343.203,171.458,51.854,160.364
C08683=1014.154,369.057,343.155,171.470,51.849,160.365
C08684=1014.161,369.305,343.116,171.480,51.846,160.366
C08685=1014.170,369.551,343.077,171.489,51.843,160.367
C08686=1014.178,369.799,343.038,171.498,51.840,160.368
C08687=1014.185,370.045,342.999,171.507,51.837,160.369
C08688=1014.193,370.292,342.960,171.517,51.833,160.370
C08689=1014.202,370.539,342.921,171.527,51.831,160.371
C08690=1014.209,370.785,342.881,171.536,51.828,160.372
C08691=1014.218,371.032,342.841,171.545,51.824,160.373
C08692=1014.225,371.279,342.803,171.555,51.822,160.374
C08693=1014.233,371.525,342.763,171.565,51.818,160.376
C08694=1014.241,371.772,342.724,171.574,51.816,160.377
C08695=1014.249,372.019,342.684,171.583,51.812,160.377
C08696=1014.258,372.266,342.645,171.593,51.809,160.378
C08697=1014.266,372.513,342.606,171.603,51.806,160.380
C08698=1014.273,372.760,342.566,171.613,51.803,160.381
C08699=1014.282,373.006,342.527,171.622,51.801,160.382
C08700=1014.290,373.253,342.488,171.632,51.797,160.383
C08701=1014.298,373.500,342.448,171.642,51.795,160.384
C08702=1014.307,373.746,342.408,171.651,51.792,160.385
C08703=1014.315,373.993,342.369,171.661,51.789,160.386
C08704=1014.323,374.240,342.329,171.671,51.786,160.387
C08705=1014.332,374.486,342.289,171.680,51.783,160.388
C08706=1014.339,374.733,342.249,171.691,51.780,160.389
C08707=1014.348,374.979,342.210,171.700,51.777,160.391
C08708=1014.356,375.226,342.170,171.709,51.774,160.392
C08709=1014.364,375.473,342.131,171.720,51.771,160.393
C08710=1014.372,375.719,342.090,171.729,51.768,160.394
C08711=1014.381,375.966,342.050,171.739,51.766,160.395
C08712=1014.389,376.213,342.010,171.749,51.763,160.396
C08713=1014.397,376.460,341.970,171.759,51.760,160.397
C08714=1014.405,376.706,341.929,171.770,51.757,160.399
C08715=1014.413,376.952,341.890,171.779,51.755,160.400
C08716=1014.421,377.199,341.849,171.788,51.752,160.401
C08717=1014.430,377.446,341.808,171.799,51.749,160.402
C08718=1014.438,377.692,341.769,171.809,51.747,160.403
C08719=1014.446,377.939,341.728,171.819,51.744,160.405
C08720=1014.454,378.185,341.687,171.829,51.741,160.406
C08721=1014.463,378.432,341.646,171.840,51.739,160.407
C08722=1014.471,378.679,341.607,171.849,51.736,160.408
C08723=1014.479,378.925,341.567,171.860,51.733,160.409
C08724=1014.488,379.172,341.526,171.869,51.730,160.411
C08725=1014.497,379.418,341.485,171.880,51.728,160.412
C08726=1014.505,379.665,341.444,171.890,51.726,160.413
C08727=1014.514,379.911,341.404,171.900,51.722,160.414
C08728=1014.522,380.157,341.363,171.910,51.720,160.416
C08729=1014.531,380.404,341.323,171.921,51.718,160.417
C08730=1014.539,380.650,341.282,171.930,51.715,160.418
C08731=1014.548,380.897,341.241,171.941,51.712,160.419
C08732=1014.556,381.143,341.201,171.951,51.710,160.421
C08733=1014.565,381.390,341.160,171.962,51.708,160.422
C08734=1014.573,381.636,341.119,171.971,51.705,160.423
C08735=1014.582,381.883,341.079,171.982,51.702,160.424
C08736=1014.591,382.130,341.037,171.992,51.700,160.426
C08737=1014.599,382.376,340.997,172.002,51.697,160.427
C08738=1014.608,382.623,340.956,172.013,51.695,160.428
C08739=1014.617,382.869,340.916,172.024,51.692,160.430
C08740=1014.626,383.115,340.874,172.034,51.690,160.431
C08741=1014.635,383.360,340.833,172.044,51.687,160.432
C08742=1014.647,383.696,340.778,172.059,51.684,160.434
C08743=1014.658,384.029,340.722,172.073,51.681,160.436
C08744=1014.670,384.365,340.667,172.087,51.678,160.438
C08745=1014.682,384.699,340.610,172.102,51.675,160.440
C08746=1014.691,384.946,340.569,172.112,51.672,160.441
C08747=1014.700,385.193,340.528,172.123,51.670,160.443
C08748=1014.709,385.439,340.486,172.134,51.668,160.444
C08749=1014.717,385.685,340.445,172.144,51.666,160.446
C08750=1014.726,385.931,340.403,172.155,51.663,160.447
C08751=1014.735,386.177,340.361,172.166,51.661,160.448
C08752=1014.744,386.424,340.320,172.177,51.659,160.450
C08753=1014.753,386.670,340.278,172.188,51.657,160.451
C08754=1014.761,386.917,340.237,172.198,51.654,160.453
C08755=1014.770,387.163,340.195,172.209,51.652,160.454
C08756=1014.779,387.410,340.153,172.220,51.650,160.456
C08757=1014.789,387.655,340.111,172.231,51.648,160.457
C08758=1014.798,387.902,340.069,172.242,51.645,160.459
C08759=1014.806,388.148,340.028,172.252,51.644,160.460
C08760=1014.815,388.395,339.986,172.263,51.642,160.462
C08761=1014.824,388.641,339.944,172.274,51.640,160.463
C08762=1014.834,388.887,339.902,172.285,51.637,160.465
C08763=1014.842,389.133,339.860,172.296,51.635,160.466
C08764=1014.851,389.380,339.818,172.308,51.633,160.468
C08765=1014.860,389.625,339.775,172.319,51.631,160.469
C08766=1014.869,389.872,339.733,172.330,51.629,160.471
C08767=1014.878,390.118,339.691,172.341,51.627,160.472
C08768=1014.887,390.364,339.649,172.352,51.625,160.474
C08769=1014.897,390.610,339.607,172.362,51.623,160.475
C08770=1014.906,390.857,339.565,172.373,51.621,160.477
C08771=1014.915,391.102,339.522,172.385,51.619,160.479
C08772=1014.924,391.349,339.481,172.396,51.617,160.480
C08773=1014.934,391.595,339.438,172.407,51.615,160.482
C08774=1014.942,391.841,339.395,172.418,51.613,160.483
C08775=1014.952,392.087,339.352,172.430,51.612,160.485
C08776=1014.960,392.333,339.311,172.442,51.609,160.487
C08777=1014.970,392.580,339.267,172.453,51.608,160.488
C08778=1014.979,392.826,339.225,172.464,51.606,160.490
C08779=1014.988,393.072,339.182,172.476,51.604,160.492
C08780=1014.998,393.318,339.140,172.487,51.602,160.493
C08781=1015.006,393.564,339.097,172.498,51.600,160.495
C08782=1015.016,393.811,339.054,172.510,51.599,160.497
C08783=1015.025,394.056,339.011,172.521,51.597,160.498
C08784=1015.036,394.302,338.968,172.533,51.595,160.500
C08785=1015.044,394.548,338.925,172.544,51.593,160.502
C08786=1014.693,392.504,338.935,172.432,51.670,160.501
C08787=1014.684,392.258,338.977,172.420,51.672,160.499
C08788=1014.675,392.012,339.019,172.409,51.674,160.498
C08789=1014.666,391.766,339.062,172.398,51.676,160.496
C08790=1014.656,391.520,339.105,172.387,51.678,160.495
C08791=1014.648,391.273,339.147,172.375,51.680,160.493
C08792=1014.638,391.028,339.189,172.364,51.682,160.491
C08793=1014.629,390.781,339.231,172.353,51.684,160.490
C08794=1014.620,390.535,339.274,172.342,51.686,160.488
C08795=1014.611,390.288,339.316,172.331,51.688,160.487
C08796=1014.601,390.043,339.358,172.319,51.690,160.485
C08797=1014.592,389.796,339.400,172.309,51.693,160.484
C08798=1014.583,389.551,339.442,172.297,51.695,160.482
C08799=1014.575,389.304,339.485,172.286,51.697,160.481
C08800=1014.566,389.058,339.526,172.275,51.699,160.479
C08801=1014.557,388.812,339.569,172.264,51.701,160.478
C08802=1014.548,388.565,339.610,172.253,51.703,160.476
C08803=1014.539,388.319,339.652,172.242,51.705,160.474
C08804=1014.530,388.073,339.694,172.232,51.707,160.473
C08805=1014.521,387.826,339.736,172.221,51.709,160.472
C08806=1014.512,387.580,339.777,172.210,51.712,160.470
C08807=1014.503,387.334,339.819,172.199,51.714,160.469
C08808=1014.494,387.087,339.861,172.188,51.717,160.467
C08809=1014.485,386.841,339.902,172.177,51.719,160.466
C08810=1014.476,386.594,339.944,172.166,51.721,160.464
C08811=1014.467,386.348,339.986,172.156,51.723,160.463
C08812=1014.459,386.102,340.028,172.145,51.725,160.461
C08813=1014.450,385.855,340.069,172.134,51.728,160.460
C08814=1014.441,385.610,340.111,172.123,51.730,160.458
C08815=1014.433,385.363,340.152,172.112,51.732,160.457
C08816=1014.424,385.116,340.193,172.102,51.735,160.456
C08817=1014.415,384.870,340.235,172.091,51.737,160.454
C08818=1014.407,384.624,340.276,172.080,51.739,160.453
C08819=1014.399,384.414,340.311,172.072,51.742,160.452
C08820=1014.391,384.204,340.346,172.062,51.744,160.451
C08821=1014.384,383.995,340.381,172.053,51.746,160.449
C08822=1014.376,383.784,340.416,172.044,51.748,160.448
C08823=1014.369,383.575,340.451,172.035,51.750,160.447
C08824=1014.361,383.366,340.486,172.026,51.752,160.446
C08825=1014.354,383.156,340.520,172.017,51.754,160.445
C08826=1014.346,382.946,340.555,172.009,51.756,160.444
C08827=1014.338,382.700,340.596,171.998,51.758,160.442
C08828=1014.329,382.453,340.638,171.987,51.762,160.441
C08829=1014.320,382.208,340.678,171.978,51.764,160.440
C08830=1014.312,381.961,340.719,171.967,51.766,160.438
C08831=1014.303,381.714,340.760,171.956,51.769,160.437
C08832=1014.294,381.468,340.800,171.946,51.771,160.436
C08833=1014.286,381.221,340.841,171.935,51.774,160.434
C08834=1014.278,380.974,340.881,171.925,51.777,160.433
C08835=1014.268,380.728,340.922,171.915,51.779,160.432
C08836=1014.260,380.481,340.962,171.904,51.782,160.431
C08837=1014.252,380.235,341.003,171.895,51.785,160.430
C08838=1014.243,379.988,341.044,171.884,51.787,160.428
C08839=1014.235,379.742,341.084,171.873,51.790,160.427
C08840=1014.226,379.495,341.125,171.864,51.793,160.426
C08841=1014.218,379.249,341.166,171.853,51.795,160.424
C08842=1014.209,379.003,341.206,171.844,51.798,160.423
C08843=1014.201,378.756,341.247,171.833,51.801,160.422
C08844=1014.193,378.509,341.287,171.824,51.803,160.421
C08845=1014.184,378.263,341.327,171.813,51.806,160.420
C08846=1014.176,378.016,341.368,171.803,51.809,160.418
C08847=1014.168,377.769,341.408,171.793,51.811,160.417
C08848=1014.160,377.523,341.448,171.783,51.814,160.416
C08849=1014.151,377.277,341.488,171.773,51.817,160.415
C08850=1014.143,377.030,341.528,171.763,51.819,160.414
C08851=1014.135,376.783,341.569,171.753,51.823,160.412
C08852=1014.126,376.536,341.609,171.743,51.826,160.411
C08853=1014.118,376.290,341.649,171.732,51.828,160.410
C08854=1014.111,376.043,341.689,171.723,51.831,160.409
C08855=1014.102,375.797,341.730,171.714,51.834,160.408
C08856=1014.094,375.550,341.769,171.703,51.837,160.407
C08857=1014.086,375.304,341.810,171.694,51.840,160.406
C08858=1014.078,375.057,341.850,171.684,51.843,160.404
C08859=1014.070,374.810,341.889,171.674,51.846,160.403
C08860=1014.061,374.563,341.929,171.664,51.849,160.402
C08861=1014.053,374.316,341.969,171.654,51.852,160.401
C08862=1014.045,374.070,342.008,171.645,51.855,160.400
C08863=1014.036,373.823,342.047,171.635,51.858,160.399
C08864=1014.028,373.576,342.087,171.625,51.861,160.398
C08865=1014.020,373.330,342.126,171.615,51.864,160.397
C08866=1014.011,373.083,342.166,171.605,51.867,160.396
C08867=1014.004,372.836,342.206,171.596,51.869,160.395
C08868=1013.995,372.589,342.245,171.586,51.873,160.393
C08869=1013.987,372.344,342.284,171.576,51.875,160.392
C08870=1013.980,372.097,342.324,171.567,51.879,160.392
C08871=1013.972,371.849,342.362,171.557,51.882,160.390
C08872=1013.964,371.603,342.402,171.547,51.885,160.389
C08873=1013.955,371.356,342.442,171.538,51.888,160.388
C08874=1013.947,371.109,342.481,171.529,51.891,160.387
C08875=1013.940,370.862,342.520,171.519,51.894,160.386
C08876=1013.932,370.616,342.559,171.510,51.898,160.385
C08877=1013.923,370.369,342.599,171.500,51.901,160.384
C08878=1013.916,370.122,342.638,171.490,51.904,160.383
C08879=1013.907,369.875,342.677,171.481,51.907,160.382
C08880=1013.901,369.628,342.716,171.472,51.910,160.381
C08881=1013.892,369.382,342.755,171.463,51.913,160.380
C08882=1013.884,369.135,342.794,171.453,51.916,160.379
C08883=1013.874,368.829,342.842,171.441,51.921,160.378
C08884=1013.864,368.524,342.891,171.430,51.924,160.377
C08885=1013.855,368.218,342.940,171.418,51.929,160.376
C08886=1013.846,367.912,342.987,171.407,51.933,160.374
C08887=1013.838,367.666,343.026,171.398,51.936,160.374
C08888=1013.830,367.419,343.065,171.388,51.939,160.373
C08889=1013.822,367.171,343.104,171.378,51.943,160.372
C08890=1013.815,366.925,343.143,171.369,51.946,160.371
C08891=1013.806,366.678,343.182,171.360,51.949,160.370
C08892=1013.799,366.432,343.220,171.351,51.952,160.369
C08893=1013.791,366.185,343.259,171.342,51.956,160.368
C08894=1013.783,365.938,343.297,171.333,51.959,160.367
C08895=1013.775,365.691,343.335,171.323,51.963,160.366
C08896=1013.768,365.444,343.373,171.314,51.966,160.365
C08897=1013.760,365.196,343.412,171.305,51.970,160.364
C08898=1013.752,364.950,343.450,171.296,51.973,160.364
C08899=1013.744,364.709,343.487,171.287,51.977,160.363
C08900=1013.738,364.468,343.525,171.278,51.980,160.362
C08901=1013.730,364.228,343.562,171.269,51.984,160.361
C08902=1013.722,363.987,343.599,171.260,51.987,160.360
C08903=1013.715,363.747,343.636,171.252,51.990,160.359
C08904=1013.707,363.506,343.674,171.243,51.994,160.359
C08905=1013.699,363.266,343.711,171.234,51.997,160.358
C08906=1013.692,363.025,343.748,171.225,52.000,160.357
C08907=1013.684,362.778,343.787,171.216,52.004,160.356
C08908=1013.677,362.531,343.824,171.208,52.008,160.355
C08909=1013.669,362.284,343.862,171.199,52.011,160.354
C08910=1013.662,362.038,343.901,171.190,52.015,160.354
C08911=1013.654,361.790,343.939,171.181,52.018,160.353
C08912=1013.646,361.544,343.977,171.172,52.022,160.352
C08913=1013.639,361.296,344.014,171.163,52.026,160.351
C08914=1013.632,361.050,344.053,171.154,52.029,160.350
C08915=1013.624,360.803,344.090,171.145,52.033,160.349
C08916=1013.617,360.555,344.128,171.137,52.037,160.349
C08917=1013.609,360.308,344.166,171.128,52.040,160.348
C08918=1013.602,360.061,344.204,171.119,52.044,160.347
C08919=1013.595,359.814,344.242,171.110,52.048,160.347
C08920=1013.588,359.567,344.280,171.101,52.051,160.346
C08921=1013.581,359.320,344.318,171.093,52.055,160.345
C08922=1013.573,359.073,344.355,171.084,52.059,160.344
C08923=1013.566,358.826,344.393,171.075,52.063,160.343
C08924=1013.558,358.579,344.431,171.066,52.066,160.343
C08925=1013.550,358.333,344.468,171.058,52.070,160.342
C08926=1013.543,358.085,344.505,171.049,52.074,160.341
C08927=1013.536,357.838,344.543,171.040,52.078,160.340
C08928=1013.529,357.591,344.580,171.032,52.082,160.340
C08929=1013.522,357.344,344.618,171.023,52.085,160.339
C08930=1013.514,357.097,344.655,171.014,52.089,160.338
C08931=1013.507,356.849,344.692,171.005,52.093,160.338
C08932=1013.499,356.602,344.729,170.996,52.097,160.337
C08933=1013.492,356.355,344.767,170.988,52.101,160.336
C08934=1013.484,356.108,344.804,170.979,52.105,160.336
C08935=1013.477,355.861,344.841,170.971,52.109,160.335
C08936=1013.470,355.614,344.879,170.962,52.113,160.334
C08937=1013.462,355.367,344.915,170.953,52.117,160.333
C08938=1013.455,355.119,344.952,170.946,52.120,160.333
C08939=1013.447,354.872,344.990,170.937,52.124,160.332
C08940=1013.441,354.625,345.027,170.929,52.129,160.332
C08941=1013.433,354.378,345.063,170.920,52.133,160.331
C08942=1013.426,354.131,345.100,170.912,52.137,160.330
C08943=1013.417,353.820,345.147,170.901,52.142,160.329
C08944=1013.408,353.510,345.194,170.890,52.146,160.329
C08945=1013.399,353.198,345.239,170.879,52.152,160.328
C08946=1013.390,352.887,345.286,170.869,52.157,160.327
C08947=1013.383,352.641,345.323,170.860,52.161,160.326
C08948=1013.375,352.394,345.359,170.853,52.165,160.326
C08949=1013.368,352.146,345.396,170.844,52.169,160.325
C08950=1013.361,351.900,345.433,170.836,52.173,160.324
C08951=1013.354,351.652,345.470,170.827,52.178,160.324
C08952=1013.346,351.404,345.506,170.819,52.182,160.323
C08953=1013.340,351.157,345.542,170.810,52.186,160.323
C08954=1013.332,350.911,345.579,170.802,52.190,160.322
C08955=1013.325,350.663,345.616,170.794,52.194,160.322
C08956=1013.318,350.416,345.652,170.786,52.199,160.321
C08957=1013.311,350.168,345.689,170.778,52.203,160.320
C08958=1013.303,349.921,345.725,170.769,52.207,160.320
C08959=1013.297,349.674,345.761,170.761,52.211,160.319
C08960=1013.289,349.426,345.797,170.752,52.216,160.319
C08961=1013.283,349.179,345.834,170.745,52.219,160.318
C08962=1013.275,348.932,345.870,170.737,52.224,160.318
C08963=1013.269,348.685,345.907,170.728,52.228,160.317
C08964=1013.261,348.437,345.943,170.720,52.233,160.317
C08965=1013.255,348.190,345.979,170.712,52.237,160.316
C08966=1013.247,347.943,346.015,170.704,52.241,160.316
C08967=1013.241,347.696,346.052,170.696,52.245,160.315
C08968=1013.235,347.449,346.088,170.687,52.249,160.314
C08969=1013.227,347.201,346.125,170.679,52.254,160.314
C08970=1013.220,346.954,346.160,170.672,52.259,160.314
C08971=1013.213,346.706,346.197,170.663,52.263,160.313
C08972=1013.206,346.459,346.232,170.655,52.267,160.312
C08973=1013.200,346.212,346.269,170.647,52.271,160.312
C08974=1013.193,345.964,346.304,170.640,52.276,160.311
C08975=1013.185,345.718,346.340,170.631,52.281,160.311
C08976=1013.179,345.470,346.376,170.623,52.285,160.310
C08977=1013.172,345.222,346.412,170.615,52.289,160.310
C08978=1013.165,344.975,346.447,170.608,52.294,160.310
C08979=1013.158,344.728,346.483,170.599,52.299,160.309
C08980=1013.151,344.480,346.519,170.591,52.303,160.308
C08981=1013.144,344.233,346.555,170.583,52.307,160.308
C08982=1013.137,343.986,346.590,170.576,52.312,160.308
C08983=1013.130,343.738,346.626,170.568,52.316,160.307
C08984=1013.124,343.491,346.662,170.559,52.321,160.307
C08985=1013.117,343.243,346.697,170.551,52.325,160.306
C08986=1013.110,342.997,346.733,170.544,52.330,160.306
C08987=1013.103,342.749,346.768,170.536,52.334,160.305
C08988=1013.096,342.501,346.804,170.527,52.339,160.305
C08989=1013.089,342.254,346.840,170.520,52.344,160.305
C08990=1013.083,342.007,346.875,170.512,52.348,160.304
C08991=1013.076,341.759,346.910,170.504,52.353,160.304
C08992=1013.069,341.512,346.946,170.496,52.358,160.303
C08993=1013.063,341.264,346.981,170.489,52.362,160.303
C08994=1013.056,341.017,347.016,170.481,52.367,160.302
C08995=1013.049,340.770,347.052,170.473,52.372,160.302
C08996=1013.042,340.523,347.087,170.465,52.376,160.302
C08997=1013.035,340.275,347.123,170.457,52.381,160.301
C08998=1013.029,340.027,347.159,170.449,52.386,160.301
C08999=1013.022,339.780,347.194,170.443,52.391,160.301
C09000=1013.016,339.532,347.229,170.434,52.395,160.300
C09001=1013.009,339.285,347.264,170.426,52.400,160.300
C09002=1013.002,339.038,347.299,170.419,52.404,160.299
C09003=1012.994,338.737,347.341,170.409,52.411,160.299
C09004=1012.987,338.437,347.384,170.400,52.416,160.298
C09005=1012.978,338.136,347.427,170.391,52.422,160.298
C09006=1012.970,337.836,347.469,170.381,52.428,160.298
C09007=1012.964,337.588,347.503,170.374,52.432,160.297
C09008=1012.957,337.340,347.539,170.366,52.438,160.297
C09009=1012.950,337.093,347.574,170.358,52.443,160.297
C09010=1012.944,336.845,347.608,170.351,52.447,160.296
C09011=1012.937,336.598,347.643,170.343,52.452,160.296
C09012=1012.930,336.350,347.678,170.335,52.457,160.296
C09013=1012.924,336.102,347.713,170.328,52.462,160.295
C09014=1012.917,335.855,347.748,170.320,52.467,160.295
C09015=1012.910,335.608,347.781,170.313,52.472,160.295
C09016=1012.903,335.360,347.817,170.306,52.477,160.294
C09017=1012.897,335.112,347.851,170.298,52.482,160.294
C09018=1012.890,334.865,347.886,170.291,52.487,160.294
C09019=1012.884,334.618,347.920,170.283,52.492,160.294
C09020=1012.878,334.370,347.955,170.275,52.497,160.293
C09021=1012.871,334.122,347.990,170.268,52.502,160.293
C09022=1012.865,333.874,348.024,170.260,52.507,160.293
C09023=1012.859,333.628,348.059,170.252,52.512,160.292
C09024=1012.852,333.380,348.093,170.246,52.517,160.292
C09025=1012.846,333.132,348.128,170.238,52.522,160.292
C09026=1012.839,332.886,348.162,170.231,52.527,160.292
C09027=1012.832,332.638,348.196,170.223,52.532,160.291
C09028=1012.826,332.390,348.231,170.215,52.537,160.291
C09029=1012.820,332.142,348.265,170.208,52.542,160.291
C09030=1012.813,331.895,348.300,170.201,52.547,160.291
C09031=1012.807,331.647,348.334,170.194,52.553,160.290
C09032=1012.800,331.400,348.368,170.186,52.557,160.290
C09033=1012.794,331.152,348.402,170.178,52.563,160.290
C09034=1012.788,330.905,348.436,170.172,52.568,160.290
C09035=1012.781,330.657,348.470,170.164,52.573,160.289
C09036=1012.774,330.409,348.505,170.156,52.579,160.289
C09037=1012.768,330.162,348.539,170.150,52.584,160.289
C09038=1012.761,329.914,348.572,170.141,52.588,160.289
C09039=1012.755,329.667,348.606,170.135,52.594,160.288
C09040=1012.749,329.419,348.641,170.127,52.599,160.288
C09041=1012.742,329.171,348.674,170.119,52.604,160.288
C09042=1012.736,328.923,348.708,170.113,52.609,160.288
C09043=1012.730,328.676,348.742,170.105,52.615,160.288
C09044=1012.723,328.428,348.776,170.098,52.620,160.287
C09045=1012.717,328.181,348.810,170.091,52.625,160.287
C09046=1012.710,327.933,348.844,170.083,52.631,160.287
C09047=1012.704,327.685,348.877,170.076,52.636,160.287
C09048=1012.698,327.438,348.911,170.069,52.641,160.287
C09049=1012.691,327.190,348.945,170.062,52.646,160.286
C09050=1012.686,326.943,348.978,170.055,52.652,160.286
C09051=1012.679,326.695,349.013,170.048,52.658,160.286
C09052=1012.673,326.448,349.046,170.040,52.663,160.286
C09053=1012.667,326.200,349.080,170.033,52.668,160.286
C09054=1012.661,325.952,349.114,170.026,52.673,160.286
C09055=1012.654,325.705,349.147,170.018,52.679,160.285
C09056=1012.648,325.457,349.181,170.012,52.685,160.286
C09057=1012.642,325.210,349.214,170.004,52.690,160.285
C09058=1012.635,324.962,349.247,169.997,52.696,160.285
C09059=1012.629,324.714,349.280,169.990,52.701,160.285
C09060=1012.622,324.466,349.313,169.983,52.707,160.285
C09061=1012.616,324.218,349.347,169.976,52.712,160.285
C09062=1012.610,323.971,349.380,169.969,52.718,160.285
C09063=1012.602,323.665,349.421,169.960,52.725,160.285
C09064=1012.594,323.361,349.461,169.951,52.731,160.284
C09065=1012.586,323.056,349.502,169.942,52.738,160.284
C09066=1012.578,322.751,349.543,169.934,52.745,160.284
C09067=1012.572,322.503,349.576,169.927,52.751,160.284
C09068=1012.566,322.256,349.609,169.919,52.756,160.284
C09069=1012.559,322.008,349.641,169.913,52.762,160.284
C09070=1012.553,321.759,349.675,169.905,52.767,160.284
C09071=1012.547,321.512,349.708,169.899,52.773,160.284
C09072=1012.540,321.264,349.741,169.891,52.779,160.283
C09073=1012.534,321.017,349.773,169.884,52.785,160.283
C09074=1012.528,320.769,349.806,169.878,52.790,160.284
C09075=1012.522,320.521,349.839,169.870,52.796,160.283
C09076=1012.516,320.274,349.872,169.864,52.802,160.283
C09077=1012.510,320.026,349.905,169.856,52.807,160.283
C09078=1012.503,319.778,349.938,169.850,52.813,160.283
C09079=1012.497,319.530,349.971,169.843,52.819,160.283
C09080=1012.490,319.283,350.004,169.835,52.824,160.283
C09081=1012.485,319.035,350.037,169.829,52.830,160.283
